ABB RobotStudio station: Final_Project.rspag

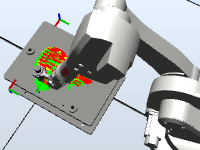
--- station ---
Station Final_Project (saved by RobotStudio 6.6.7603.115)
Controller IRB_1600_8kg_1.45m
  mechanical unit ROB_1: IRB1600_8_145__02, 6 joints, base frame (0, 0, 0) mm
Layout (positions relative to the parent item):
  - IRB1600_8_145__02 [mechanism, from Robots\IRB1600_8_145_G_02.rslib] at (0, 0, 0) mm; joint values [0.2552, 0.6803, 0.4832, 0.5846, -0.2854, -0.363] (rad or m)
  - Robotpedestal1400_H240 [part, from Equipment\Robot Pedestal 1400 H240.rslib] at (876.55, 58.92, 0) mm
  - MyTool [mechanism, from Training Objects\myTool.rslib] at (841.22, 209, 428.53) mm, rotated rx 180 ry 38 rz 180 deg
Attachment: MyTool is attached to IRB1600_8_145__02 / Link6

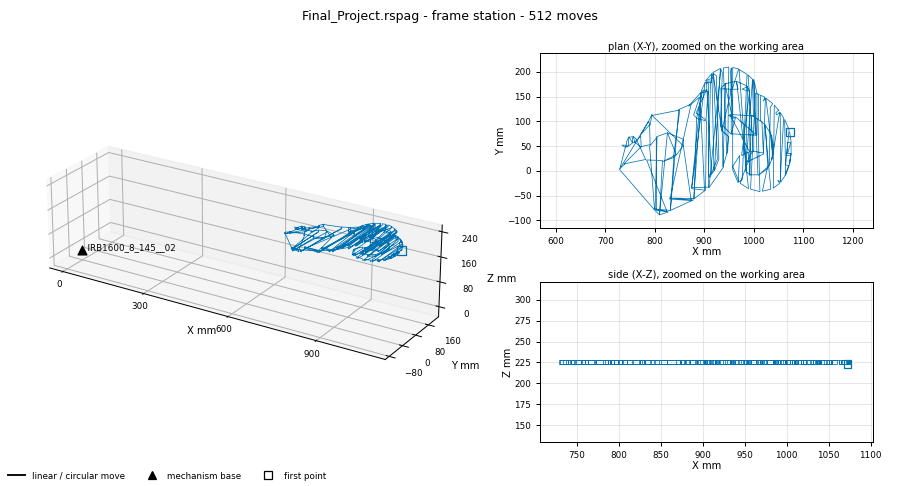
[picture p0: tool path of Final_Project.rspag in frame station, 512 of 512 moves have a stored position in this frame; points joined in program order, loops and branches not executed]
--- Backups/IRB_1600_8kg_1.45m/RAPID/TASK1/PROGMOD/CalibData.mod ---
MODULE CalibData
	TASK PERS wobjdata Workobject_1:=[FALSE,TRUE,"",[[1116.549,-245,225],[0.707106781,0,0,0.707106781]],[[600,0,8],[0,0,1,0]]];
	TASK PERS tooldata MyTool:=[TRUE,[[31.792631019,0,229.638935148],[0.945518576,0,0.325568154,0]],[1,[0,0,1],[1,0,0,0],0,0,0]];
ENDMODULE

--- Backups/IRB_1600_8kg_1.45m/RAPID/TASK1/PROGMOD/Module1.mod ---
MODULE Module1
    CONST robtarget point_0_clearance:=[[277,44,10],[0.707106781,0,0,0.707106781],[0,0,-1,1],[9E+09,9E+09,9E+09,9E+09,9E+09,9E+09]];
    CONST robtarget point_0_contact:=[[277,44,5],[0.707106781,0,0,0.707106781],[0,0,-1,1],[9E+09,9E+09,9E+09,9E+09,9E+09,9E+09]];
    CONST robtarget point_1_contact:=[[296,41,5],[0.707106781,0,0,0.707106781],[0,0,-1,1],[9E+09,9E+09,9E+09,9E+09,9E+09,9E+09]];
    CONST robtarget point_1_clearance:=[[296,41,10],[0.707106781,0,0,0.707106781],[0,0,-1,1],[9E+09,9E+09,9E+09,9E+09,9E+09,9E+09]];
    CONST robtarget point_2_clearance:=[[322,41,10],[0.707106781,0,0,0.707106781],[0,0,-1,1],[9E+09,9E+09,9E+09,9E+09,9E+09,9E+09]];
    CONST robtarget point_2_contact:=[[322,41,5],[0.707106781,0,0,0.707106781],[0,0,-1,1],[9E+09,9E+09,9E+09,9E+09,9E+09,9E+09]];
    CONST robtarget point_3_contact:=[[341,44,5],[0.707106781,0,0,0.707106781],[0,0,-1,1],[9E+09,9E+09,9E+09,9E+09,9E+09,9E+09]];
    CONST robtarget point_3_clearance:=[[341,44,10],[0.707106781,0,0,0.707106781],[0,0,-1,1],[9E+09,9E+09,9E+09,9E+09,9E+09,9E+09]];
    CONST robtarget point_4_clearance:=[[320,41,10],[0.707106781,0,0,0.707106781],[0,0,-1,1],[9E+09,9E+09,9E+09,9E+09,9E+09,9E+09]];
    CONST robtarget point_4_contact:=[[320,41,5],[0.707106781,0,0,0.707106781],[0,0,-1,1],[9E+09,9E+09,9E+09,9E+09,9E+09,9E+09]];
    CONST robtarget point_5_contact:=[[320,48,5],[0.707106781,0,0,0.707106781],[0,0,-1,1],[9E+09,9E+09,9E+09,9E+09,9E+09,9E+09]];
    CONST robtarget point_5_clearance:=[[320,48,10],[0.707106781,0,0,0.707106781],[0,0,-1,1],[9E+09,9E+09,9E+09,9E+09,9E+09,9E+09]];
    CONST robtarget point_6_clearance:=[[298,42,10],[0.707106781,0,0,0.707106781],[0,0,-1,1],[9E+09,9E+09,9E+09,9E+09,9E+09,9E+09]];
    CONST robtarget point_6_contact:=[[298,42,5],[0.707106781,0,0,0.707106781],[0,0,-1,1],[9E+09,9E+09,9E+09,9E+09,9E+09,9E+09]];
    CONST robtarget point_7_contact:=[[298,48,5],[0.707106781,0,0,0.707106781],[0,0,-1,1],[9E+09,9E+09,9E+09,9E+09,9E+09,9E+09]];
    CONST robtarget point_7_clearance:=[[298,48,10],[0.707106781,0,0,0.707106781],[0,0,-1,1],[9E+09,9E+09,9E+09,9E+09,9E+09,9E+09]];
    CONST robtarget point_8_clearance:=[[324,50,10],[0.707106781,0,0,0.707106781],[0,0,-1,1],[9E+09,9E+09,9E+09,9E+09,9E+09,9E+09]];
    CONST robtarget point_8_contact:=[[324,50,5],[0.707106781,0,0,0.707106781],[0,0,-1,1],[9E+09,9E+09,9E+09,9E+09,9E+09,9E+09]];
    CONST robtarget point_9_contact:=[[323,42,5],[0.707106781,0,0,0.707106781],[0,0,-1,1],[9E+09,9E+09,9E+09,9E+09,9E+09,9E+09]];
    CONST robtarget point_9_clearance:=[[323,42,10],[0.707106781,0,0,0.707106781],[0,0,-1,1],[9E+09,9E+09,9E+09,9E+09,9E+09,9E+09]];
    CONST robtarget point_10_clearance:=[[345,45,10],[0.707106781,0,0,0.707106781],[0,0,-1,1],[9E+09,9E+09,9E+09,9E+09,9E+09,9E+09]];
    CONST robtarget point_10_contact:=[[345,45,5],[0.707106781,0,0,0.707106781],[0,0,-1,1],[9E+09,9E+09,9E+09,9E+09,9E+09,9E+09]];
    CONST robtarget point_11_contact:=[[364,52,5],[0.707106781,0,0,0.707106781],[-1,-1,0,1],[9E+09,9E+09,9E+09,9E+09,9E+09,9E+09]];
    CONST robtarget point_11_clearance:=[[364,52,10],[0.707106781,0,0,0.707106781],[-1,-1,0,1],[9E+09,9E+09,9E+09,9E+09,9E+09,9E+09]];
    CONST robtarget point_12_clearance:=[[251,54,10],[0.707106781,0,0,0.707106781],[0,0,-1,1],[9E+09,9E+09,9E+09,9E+09,9E+09,9E+09]];
    CONST robtarget point_12_contact:=[[251,54,5],[0.707106781,0,0,0.707106781],[0,0,-1,1],[9E+09,9E+09,9E+09,9E+09,9E+09,9E+09]];
    CONST robtarget point_13_contact:=[[272,45,5],[0.707106781,0,0,0.707106781],[0,0,-1,1],[9E+09,9E+09,9E+09,9E+09,9E+09,9E+09]];
    CONST robtarget point_13_clearance:=[[272,45,10],[0.707106781,0,0,0.707106781],[0,0,-1,1],[9E+09,9E+09,9E+09,9E+09,9E+09,9E+09]];
    CONST robtarget point_14_clearance:=[[343,52,10],[0.707106781,0,0,0.707106781],[0,0,-1,1],[9E+09,9E+09,9E+09,9E+09,9E+09,9E+09]];
    CONST robtarget point_14_contact:=[[343,52,5],[0.707106781,0,0,0.707106781],[0,0,-1,1],[9E+09,9E+09,9E+09,9E+09,9E+09,9E+09]];
    CONST robtarget point_15_contact:=[[344,46,5],[0.707106781,0,0,0.707106781],[0,0,-1,1],[9E+09,9E+09,9E+09,9E+09,9E+09,9E+09]];
    CONST robtarget point_15_clearance:=[[344,46,10],[0.707106781,0,0,0.707106781],[0,0,-1,1],[9E+09,9E+09,9E+09,9E+09,9E+09,9E+09]];
    CONST robtarget point_16_clearance:=[[366,54,10],[0.707106781,0,0,0.707106781],[-1,-1,0,1],[9E+09,9E+09,9E+09,9E+09,9E+09,9E+09]];
    CONST robtarget point_16_contact:=[[366,54,5],[0.707106781,0,0,0.707106781],[-1,-1,0,1],[9E+09,9E+09,9E+09,9E+09,9E+09,9E+09]];
    CONST robtarget point_17_contact:=[[378,62,5],[0.707106781,0,0,0.707106781],[-1,-1,0,1],[9E+09,9E+09,9E+09,9E+09,9E+09,9E+09]];
    CONST robtarget point_17_clearance:=[[378,62,10],[0.707106781,0,0,0.707106781],[-1,-1,0,1],[9E+09,9E+09,9E+09,9E+09,9E+09,9E+09]];
    CONST robtarget point_18_clearance:=[[237,63,10],[0.707106781,0,0,0.707106781],[0,0,-1,1],[9E+09,9E+09,9E+09,9E+09,9E+09,9E+09]];
    CONST robtarget point_18_contact:=[[237,63,5],[0.707106781,0,0,0.707106781],[0,0,-1,1],[9E+09,9E+09,9E+09,9E+09,9E+09,9E+09]];
    CONST robtarget point_19_contact:=[[248,56,5],[0.707106781,0,0,0.707106781],[0,0,-1,1],[9E+09,9E+09,9E+09,9E+09,9E+09,9E+09]];
    CONST robtarget point_19_clearance:=[[248,56,10],[0.707106781,0,0,0.707106781],[0,0,-1,1],[9E+09,9E+09,9E+09,9E+09,9E+09,9E+09]];
    CONST robtarget point_20_clearance:=[[377,63,10],[0.707106781,0,0,0.707106781],[-1,-1,0,1],[9E+09,9E+09,9E+09,9E+09,9E+09,9E+09]];
    CONST robtarget point_20_contact:=[[377,63,5],[0.707106781,0,0,0.707106781],[-1,-1,0,1],[9E+09,9E+09,9E+09,9E+09,9E+09,9E+09]];
    CONST robtarget point_21_contact:=[[374,68,5],[0.707106781,0,0,0.707106781],[-1,-1,0,1],[9E+09,9E+09,9E+09,9E+09,9E+09,9E+09]];
    CONST robtarget point_21_clearance:=[[374,68,10],[0.707106781,0,0,0.707106781],[-1,-1,0,1],[9E+09,9E+09,9E+09,9E+09,9E+09,9E+09]];
    CONST robtarget point_22_clearance:=[[380,64,10],[0.707106781,0,0,0.707106781],[-1,-1,0,1],[9E+09,9E+09,9E+09,9E+09,9E+09,9E+09]];
    CONST robtarget point_22_contact:=[[380,64,5],[0.707106781,0,0,0.707106781],[-1,-1,0,1],[9E+09,9E+09,9E+09,9E+09,9E+09,9E+09]];
    CONST robtarget point_23_contact:=[[390,77,5],[0.707106781,0,0,0.707106781],[-1,-1,0,1],[9E+09,9E+09,9E+09,9E+09,9E+09,9E+09]];
    CONST robtarget point_23_clearance:=[[390,77,10],[0.707106781,0,0,0.707106781],[-1,-1,0,1],[9E+09,9E+09,9E+09,9E+09,9E+09,9E+09]];
    CONST robtarget point_24_clearance:=[[222,75,10],[0.707106781,0,0,0.707106781],[0,0,-1,1],[9E+09,9E+09,9E+09,9E+09,9E+09,9E+09]];
    CONST robtarget point_24_contact:=[[222,75,5],[0.707106781,0,0,0.707106781],[0,0,-1,1],[9E+09,9E+09,9E+09,9E+09,9E+09,9E+09]];
    CONST robtarget point_25_contact:=[[233,66,5],[0.707106781,0,0,0.707106781],[0,0,-1,1],[9E+09,9E+09,9E+09,9E+09,9E+09,9E+09]];
    CONST robtarget point_25_clearance:=[[233,66,10],[0.707106781,0,0,0.707106781],[0,0,-1,1],[9E+09,9E+09,9E+09,9E+09,9E+09,9E+09]];
    CONST robtarget point_26_clearance:=[[232,66,10],[0.707106781,0,0,0.707106781],[0,0,-1,1],[9E+09,9E+09,9E+09,9E+09,9E+09,9E+09]];
    CONST robtarget point_26_contact:=[[232,66,5],[0.707106781,0,0,0.707106781],[0,0,-1,1],[9E+09,9E+09,9E+09,9E+09,9E+09,9E+09]];
    CONST robtarget point_27_contact:=[[238,72,5],[0.707106781,0,0,0.707106781],[0,0,-1,1],[9E+09,9E+09,9E+09,9E+09,9E+09,9E+09]];
    CONST robtarget point_27_clearance:=[[238,72,10],[0.707106781,0,0,0.707106781],[0,0,-1,1],[9E+09,9E+09,9E+09,9E+09,9E+09,9E+09]];
    CONST robtarget point_28_clearance:=[[242,70,10],[0.707106781,0,0,0.707106781],[0,0,-1,1],[9E+09,9E+09,9E+09,9E+09,9E+09,9E+09]];
    CONST robtarget point_28_contact:=[[242,70,5],[0.707106781,0,0,0.707106781],[0,0,-1,1],[9E+09,9E+09,9E+09,9E+09,9E+09,9E+09]];
    CONST robtarget point_29_contact:=[[236,64,5],[0.707106781,0,0,0.707106781],[0,0,-1,1],[9E+09,9E+09,9E+09,9E+09,9E+09,9E+09]];
    CONST robtarget point_29_clearance:=[[236,64,10],[0.707106781,0,0,0.707106781],[0,0,-1,1],[9E+09,9E+09,9E+09,9E+09,9E+09,9E+09]];
    CONST robtarget point_30_clearance:=[[310,76,10],[0.707106781,0,0,0.707106781],[0,0,-1,1],[9E+09,9E+09,9E+09,9E+09,9E+09,9E+09]];
    CONST robtarget point_30_contact:=[[310,76,5],[0.707106781,0,0,0.707106781],[0,0,-1,1],[9E+09,9E+09,9E+09,9E+09,9E+09,9E+09]];
    CONST robtarget point_31_contact:=[[283,81,5],[0.707106781,0,0,0.707106781],[0,0,-1,1],[9E+09,9E+09,9E+09,9E+09,9E+09,9E+09]];
    CONST robtarget point_31_clearance:=[[283,81,10],[0.707106781,0,0,0.707106781],[0,0,-1,1],[9E+09,9E+09,9E+09,9E+09,9E+09,9E+09]];
    CONST robtarget point_32_clearance:=[[323,78,10],[0.707106781,0,0,0.707106781],[0,0,-1,1],[9E+09,9E+09,9E+09,9E+09,9E+09,9E+09]];
    CONST robtarget point_32_contact:=[[323,78,5],[0.707106781,0,0,0.707106781],[0,0,-1,1],[9E+09,9E+09,9E+09,9E+09,9E+09,9E+09]];
    CONST robtarget point_33_contact:=[[310,77,5],[0.707106781,0,0,0.707106781],[0,0,-1,1],[9E+09,9E+09,9E+09,9E+09,9E+09,9E+09]];
    CONST robtarget point_33_clearance:=[[310,77,10],[0.707106781,0,0,0.707106781],[0,0,-1,1],[9E+09,9E+09,9E+09,9E+09,9E+09,9E+09]];
    CONST robtarget point_34_clearance:=[[332,80,10],[0.707106781,0,0,0.707106781],[0,0,-1,1],[9E+09,9E+09,9E+09,9E+09,9E+09,9E+09]];
    CONST robtarget point_34_contact:=[[332,80,5],[0.707106781,0,0,0.707106781],[0,0,-1,1],[9E+09,9E+09,9E+09,9E+09,9E+09,9E+09]];
    CONST robtarget point_35_contact:=[[321,78,5],[0.707106781,0,0,0.707106781],[0,0,-1,1],[9E+09,9E+09,9E+09,9E+09,9E+09,9E+09]];
    CONST robtarget point_35_clearance:=[[321,78,10],[0.707106781,0,0,0.707106781],[0,0,-1,1],[9E+09,9E+09,9E+09,9E+09,9E+09,9E+09]];
    CONST robtarget point_36_clearance:=[[208,92,10],[0.707106781,0,0,0.707106781],[0,0,-1,1],[9E+09,9E+09,9E+09,9E+09,9E+09,9E+09]];
    CONST robtarget point_36_contact:=[[208,92,5],[0.707106781,0,0,0.707106781],[0,0,-1,1],[9E+09,9E+09,9E+09,9E+09,9E+09,9E+09]];
    CONST robtarget point_37_contact:=[[219,78,5],[0.707106781,0,0,0.707106781],[0,0,-1,1],[9E+09,9E+09,9E+09,9E+09,9E+09,9E+09]];
    CONST robtarget point_37_clearance:=[[219,78,10],[0.707106781,0,0,0.707106781],[0,0,-1,1],[9E+09,9E+09,9E+09,9E+09,9E+09,9E+09]];
    CONST robtarget point_38_clearance:=[[219,78,10],[0.707106781,0,0,0.707106781],[0,0,-1,1],[9E+09,9E+09,9E+09,9E+09,9E+09,9E+09]];
    CONST robtarget point_38_contact:=[[219,78,5],[0.707106781,0,0,0.707106781],[0,0,-1,1],[9E+09,9E+09,9E+09,9E+09,9E+09,9E+09]];
    CONST robtarget point_39_contact:=[[226,83,5],[0.707106781,0,0,0.707106781],[0,0,-1,1],[9E+09,9E+09,9E+09,9E+09,9E+09,9E+09]];
    CONST robtarget point_39_clearance:=[[226,83,10],[0.707106781,0,0,0.707106781],[0,0,-1,1],[9E+09,9E+09,9E+09,9E+09,9E+09,9E+09]];
    CONST robtarget point_40_clearance:=[[344,85,10],[0.707106781,0,0,0.707106781],[0,0,-1,1],[9E+09,9E+09,9E+09,9E+09,9E+09,9E+09]];
    CONST robtarget point_40_contact:=[[344,85,5],[0.707106781,0,0,0.707106781],[0,0,-1,1],[9E+09,9E+09,9E+09,9E+09,9E+09,9E+09]];
    CONST robtarget point_41_contact:=[[329,79,5],[0.707106781,0,0,0.707106781],[0,0,-1,1],[9E+09,9E+09,9E+09,9E+09,9E+09,9E+09]];
    CONST robtarget point_41_clearance:=[[329,79,10],[0.707106781,0,0,0.707106781],[0,0,-1,1],[9E+09,9E+09,9E+09,9E+09,9E+09,9E+09]];
    CONST robtarget point_42_clearance:=[[284,80,10],[0.707106781,0,0,0.707106781],[0,0,-1,1],[9E+09,9E+09,9E+09,9E+09,9E+09,9E+09]];
    CONST robtarget point_42_contact:=[[284,80,5],[0.707106781,0,0,0.707106781],[0,0,-1,1],[9E+09,9E+09,9E+09,9E+09,9E+09,9E+09]];
    CONST robtarget point_43_contact:=[[261,94,5],[0.707106781,0,0,0.707106781],[0,0,-1,1],[9E+09,9E+09,9E+09,9E+09,9E+09,9E+09]];
    CONST robtarget point_43_clearance:=[[261,94,10],[0.707106781,0,0,0.707106781],[0,0,-1,1],[9E+09,9E+09,9E+09,9E+09,9E+09,9E+09]];
    CONST robtarget point_44_clearance:=[[392,82,10],[0.707106781,0,0,0.707106781],[-1,-1,0,1],[9E+09,9E+09,9E+09,9E+09,9E+09,9E+09]];
    CONST robtarget point_44_contact:=[[392,82,5],[0.707106781,0,0,0.707106781],[-1,-1,0,1],[9E+09,9E+09,9E+09,9E+09,9E+09,9E+09]];
    CONST robtarget point_45_contact:=[[396,99,5],[0.707106781,0,0,0.707106781],[-1,-1,0,1],[9E+09,9E+09,9E+09,9E+09,9E+09,9E+09]];
    CONST robtarget point_45_clearance:=[[396,99,10],[0.707106781,0,0,0.707106781],[-1,-1,0,1],[9E+09,9E+09,9E+09,9E+09,9E+09,9E+09]];
    CONST robtarget point_46_clearance:=[[349,89,10],[0.707106781,0,0,0.707106781],[0,0,-1,1],[9E+09,9E+09,9E+09,9E+09,9E+09,9E+09]];
    CONST robtarget point_46_contact:=[[349,89,5],[0.707106781,0,0,0.707106781],[0,0,-1,1],[9E+09,9E+09,9E+09,9E+09,9E+09,9E+09]];
    CONST robtarget point_47_contact:=[[344,85,5],[0.707106781,0,0,0.707106781],[0,0,-1,1],[9E+09,9E+09,9E+09,9E+09,9E+09,9E+09]];
    CONST robtarget point_47_clearance:=[[344,85,10],[0.707106781,0,0,0.707106781],[0,0,-1,1],[9E+09,9E+09,9E+09,9E+09,9E+09,9E+09]];
    CONST robtarget point_48_clearance:=[[364,107,10],[0.707106781,0,0,0.707106781],[-1,-1,0,1],[9E+09,9E+09,9E+09,9E+09,9E+09,9E+09]];
    CONST robtarget point_48_contact:=[[364,107,5],[0.707106781,0,0,0.707106781],[-1,-1,0,1],[9E+09,9E+09,9E+09,9E+09,9E+09,9E+09]];
    CONST robtarget point_49_contact:=[[350,88,5],[0.707106781,0,0,0.707106781],[0,0,-1,1],[9E+09,9E+09,9E+09,9E+09,9E+09,9E+09]];
    CONST robtarget point_49_clearance:=[[350,88,10],[0.707106781,0,0,0.707106781],[0,0,-1,1],[9E+09,9E+09,9E+09,9E+09,9E+09,9E+09]];
    CONST robtarget point_50_clearance:=[[263,93,10],[0.707106781,0,0,0.707106781],[0,0,-1,1],[9E+09,9E+09,9E+09,9E+09,9E+09,9E+09]];
    CONST robtarget point_50_contact:=[[263,93,5],[0.707106781,0,0,0.707106781],[0,0,-1,1],[9E+09,9E+09,9E+09,9E+09,9E+09,9E+09]];
    CONST robtarget point_51_contact:=[[253,103,5],[0.707106781,0,0,0.707106781],[0,0,-1,1],[9E+09,9E+09,9E+09,9E+09,9E+09,9E+09]];
    CONST robtarget point_51_clearance:=[[253,103,10],[0.707106781,0,0,0.707106781],[0,0,-1,1],[9E+09,9E+09,9E+09,9E+09,9E+09,9E+09]];
    CONST robtarget point_52_clearance:=[[202,103,10],[0.707106781,0,0,0.707106781],[0,0,-1,1],[9E+09,9E+09,9E+09,9E+09,9E+09,9E+09]];
    CONST robtarget point_52_contact:=[[202,103,5],[0.707106781,0,0,0.707106781],[0,0,-1,1],[9E+09,9E+09,9E+09,9E+09,9E+09,9E+09]];
    CONST robtarget point_53_contact:=[[206,94,5],[0.707106781,0,0,0.707106781],[0,0,-1,1],[9E+09,9E+09,9E+09,9E+09,9E+09,9E+09]];
    CONST robtarget point_53_clearance:=[[206,94,10],[0.707106781,0,0,0.707106781],[0,0,-1,1],[9E+09,9E+09,9E+09,9E+09,9E+09,9E+09]];
    CONST robtarget point_54_clearance:=[[214,97,10],[0.707106781,0,0,0.707106781],[0,0,-1,1],[9E+09,9E+09,9E+09,9E+09,9E+09,9E+09]];
    CONST robtarget point_54_contact:=[[214,97,5],[0.707106781,0,0,0.707106781],[0,0,-1,1],[9E+09,9E+09,9E+09,9E+09,9E+09,9E+09]];
    CONST robtarget point_55_contact:=[[208,93,5],[0.707106781,0,0,0.707106781],[0,0,-1,1],[9E+09,9E+09,9E+09,9E+09,9E+09,9E+09]];
    CONST robtarget point_55_clearance:=[[208,93,10],[0.707106781,0,0,0.707106781],[0,0,-1,1],[9E+09,9E+09,9E+09,9E+09,9E+09,9E+09]];
    CONST robtarget point_56_clearance:=[[321,97,10],[0.707106781,0,0,0.707106781],[0,0,-1,1],[9E+09,9E+09,9E+09,9E+09,9E+09,9E+09]];
    CONST robtarget point_56_contact:=[[321,97,5],[0.707106781,0,0,0.707106781],[0,0,-1,1],[9E+09,9E+09,9E+09,9E+09,9E+09,9E+09]];
    CONST robtarget point_57_contact:=[[337,130,5],[0.707106781,0,0,0.707106781],[0,0,-1,1],[9E+09,9E+09,9E+09,9E+09,9E+09,9E+09]];
    CONST robtarget point_57_clearance:=[[337,130,10],[0.707106781,0,0,0.707106781],[0,0,-1,1],[9E+09,9E+09,9E+09,9E+09,9E+09,9E+09]];
    CONST robtarget point_58_clearance:=[[315,119,10],[0.707106781,0,0,0.707106781],[0,0,-1,1],[9E+09,9E+09,9E+09,9E+09,9E+09,9E+09]];
    CONST robtarget point_58_contact:=[[315,119,5],[0.707106781,0,0,0.707106781],[0,0,-1,1],[9E+09,9E+09,9E+09,9E+09,9E+09,9E+09]];
    CONST robtarget point_59_contact:=[[319,97,5],[0.707106781,0,0,0.707106781],[0,0,-1,1],[9E+09,9E+09,9E+09,9E+09,9E+09,9E+09]];
    CONST robtarget point_59_clearance:=[[319,97,10],[0.707106781,0,0,0.707106781],[0,0,-1,1],[9E+09,9E+09,9E+09,9E+09,9E+09,9E+09]];
    CONST robtarget point_60_clearance:=[[256,100,10],[0.707106781,0,0,0.707106781],[0,0,-1,1],[9E+09,9E+09,9E+09,9E+09,9E+09,9E+09]];
    CONST robtarget point_60_contact:=[[256,100,5],[0.707106781,0,0,0.707106781],[0,0,-1,1],[9E+09,9E+09,9E+09,9E+09,9E+09,9E+09]];
    CONST robtarget point_61_contact:=[[251,108,5],[0.707106781,0,0,0.707106781],[0,0,-1,1],[9E+09,9E+09,9E+09,9E+09,9E+09,9E+09]];
    CONST robtarget point_61_clearance:=[[251,108,10],[0.707106781,0,0,0.707106781],[0,0,-1,1],[9E+09,9E+09,9E+09,9E+09,9E+09,9E+09]];
    CONST robtarget point_62_clearance:=[[397,104,10],[0.707106781,0,0,0.707106781],[-1,-1,0,1],[9E+09,9E+09,9E+09,9E+09,9E+09,9E+09]];
    CONST robtarget point_62_contact:=[[397,104,5],[0.707106781,0,0,0.707106781],[-1,-1,0,1],[9E+09,9E+09,9E+09,9E+09,9E+09,9E+09]];
    CONST robtarget point_63_contact:=[[392,123,5],[0.707106781,0,0,0.707106781],[-1,-1,0,1],[9E+09,9E+09,9E+09,9E+09,9E+09,9E+09]];
    CONST robtarget point_63_clearance:=[[392,123,10],[0.707106781,0,0,0.707106781],[-1,-1,0,1],[9E+09,9E+09,9E+09,9E+09,9E+09,9E+09]];
    CONST robtarget point_64_clearance:=[[198,113,10],[0.707106781,0,0,0.707106781],[0,0,-1,1],[9E+09,9E+09,9E+09,9E+09,9E+09,9E+09]];
    CONST robtarget point_64_contact:=[[198,113,5],[0.707106781,0,0,0.707106781],[0,0,-1,1],[9E+09,9E+09,9E+09,9E+09,9E+09,9E+09]];
    CONST robtarget point_65_contact:=[[201,105,5],[0.707106781,0,0,0.707106781],[0,0,-1,1],[9E+09,9E+09,9E+09,9E+09,9E+09,9E+09]];
    CONST robtarget point_65_clearance:=[[201,105,10],[0.707106781,0,0,0.707106781],[0,0,-1,1],[9E+09,9E+09,9E+09,9E+09,9E+09,9E+09]];
    CONST robtarget point_66_clearance:=[[202,107,10],[0.707106781,0,0,0.707106781],[0,0,-1,1],[9E+09,9E+09,9E+09,9E+09,9E+09,9E+09]];
    CONST robtarget point_66_contact:=[[202,107,5],[0.707106781,0,0,0.707106781],[0,0,-1,1],[9E+09,9E+09,9E+09,9E+09,9E+09,9E+09]];
    CONST robtarget point_67_contact:=[[208,107,5],[0.707106781,0,0,0.707106781],[0,0,-1,1],[9E+09,9E+09,9E+09,9E+09,9E+09,9E+09]];
    CONST robtarget point_67_clearance:=[[208,107,10],[0.707106781,0,0,0.707106781],[0,0,-1,1],[9E+09,9E+09,9E+09,9E+09,9E+09,9E+09]];
    CONST robtarget point_68_clearance:=[[251,107,10],[0.707106781,0,0,0.707106781],[0,0,-1,1],[9E+09,9E+09,9E+09,9E+09,9E+09,9E+09]];
    CONST robtarget point_68_contact:=[[251,107,5],[0.707106781,0,0,0.707106781],[0,0,-1,1],[9E+09,9E+09,9E+09,9E+09,9E+09,9E+09]];
    CONST robtarget point_69_contact:=[[243,121,5],[0.707106781,0,0,0.707106781],[0,0,-1,1],[9E+09,9E+09,9E+09,9E+09,9E+09,9E+09]];
    CONST robtarget point_69_clearance:=[[243,121,10],[0.707106781,0,0,0.707106781],[0,0,-1,1],[9E+09,9E+09,9E+09,9E+09,9E+09,9E+09]];
    CONST robtarget point_70_clearance:=[[363,125,10],[0.707106781,0,0,0.707106781],[-1,-1,0,1],[9E+09,9E+09,9E+09,9E+09,9E+09,9E+09]];
    CONST robtarget point_70_contact:=[[363,125,5],[0.707106781,0,0,0.707106781],[-1,-1,0,1],[9E+09,9E+09,9E+09,9E+09,9E+09,9E+09]];
    CONST robtarget point_71_contact:=[[363,108,5],[0.707106781,0,0,0.707106781],[-1,-1,0,1],[9E+09,9E+09,9E+09,9E+09,9E+09,9E+09]];
    CONST robtarget point_71_clearance:=[[363,108,10],[0.707106781,0,0,0.707106781],[-1,-1,0,1],[9E+09,9E+09,9E+09,9E+09,9E+09,9E+09]];
    CONST robtarget point_72_clearance:=[[172,116,10],[0.707106781,0,0,0.707106781],[0,0,-1,1],[9E+09,9E+09,9E+09,9E+09,9E+09,9E+09]];
    CONST robtarget point_72_contact:=[[172,116,5],[0.707106781,0,0,0.707106781],[0,0,-1,1],[9E+09,9E+09,9E+09,9E+09,9E+09,9E+09]];
    CONST robtarget point_73_contact:=[[198,110,5],[0.707106781,0,0,0.707106781],[0,0,-1,1],[9E+09,9E+09,9E+09,9E+09,9E+09,9E+09]];
    CONST robtarget point_73_clearance:=[[198,110,10],[0.707106781,0,0,0.707106781],[0,0,-1,1],[9E+09,9E+09,9E+09,9E+09,9E+09,9E+09]];
    CONST robtarget point_74_clearance:=[[283,110,10],[0.707106781,0,0,0.707106781],[0,0,-1,1],[9E+09,9E+09,9E+09,9E+09,9E+09,9E+09]];
    CONST robtarget point_74_contact:=[[283,110,5],[0.707106781,0,0,0.707106781],[0,0,-1,1],[9E+09,9E+09,9E+09,9E+09,9E+09,9E+09]];
    CONST robtarget point_75_contact:=[[280,162,5],[0.707106781,0,0,0.707106781],[0,0,-1,1],[9E+09,9E+09,9E+09,9E+09,9E+09,9E+09]];
    CONST robtarget point_75_clearance:=[[280,162,10],[0.707106781,0,0,0.707106781],[0,0,-1,1],[9E+09,9E+09,9E+09,9E+09,9E+09,9E+09]];
    CONST robtarget point_76_clearance:=[[246,153,10],[0.707106781,0,0,0.707106781],[0,0,-1,1],[9E+09,9E+09,9E+09,9E+09,9E+09,9E+09]];
    CONST robtarget point_76_contact:=[[246,153,5],[0.707106781,0,0,0.707106781],[0,0,-1,1],[9E+09,9E+09,9E+09,9E+09,9E+09,9E+09]];
    CONST robtarget point_77_contact:=[[281,113,5],[0.707106781,0,0,0.707106781],[0,0,-1,1],[9E+09,9E+09,9E+09,9E+09,9E+09,9E+09]];
    CONST robtarget point_77_clearance:=[[281,113,10],[0.707106781,0,0,0.707106781],[0,0,-1,1],[9E+09,9E+09,9E+09,9E+09,9E+09,9E+09]];
    CONST robtarget point_78_clearance:=[[170,117,10],[0.707106781,0,0,0.707106781],[0,0,-1,1],[9E+09,9E+09,9E+09,9E+09,9E+09,9E+09]];
    CONST robtarget point_78_contact:=[[170,117,5],[0.707106781,0,0,0.707106781],[0,0,-1,1],[9E+09,9E+09,9E+09,9E+09,9E+09,9E+09]];
    CONST robtarget point_79_contact:=[[173,119,5],[0.707106781,0,0,0.707106781],[0,0,-1,1],[9E+09,9E+09,9E+09,9E+09,9E+09,9E+09]];
    CONST robtarget point_79_clearance:=[[173,119,10],[0.707106781,0,0,0.707106781],[0,0,-1,1],[9E+09,9E+09,9E+09,9E+09,9E+09,9E+09]];
    CONST robtarget point_80_clearance:=[[244,117,10],[0.707106781,0,0,0.707106781],[0,0,-1,1],[9E+09,9E+09,9E+09,9E+09,9E+09,9E+09]];
    CONST robtarget point_80_contact:=[[244,117,5],[0.707106781,0,0,0.707106781],[0,0,-1,1],[9E+09,9E+09,9E+09,9E+09,9E+09,9E+09]];
    CONST robtarget point_81_contact:=[[241,165,5],[0.707106781,0,0,0.707106781],[0,0,-1,1],[9E+09,9E+09,9E+09,9E+09,9E+09,9E+09]];
    CONST robtarget point_81_clearance:=[[241,165,10],[0.707106781,0,0,0.707106781],[0,0,-1,1],[9E+09,9E+09,9E+09,9E+09,9E+09,9E+09]];
    CONST robtarget point_82_clearance:=[[316,125,10],[0.707106781,0,0,0.707106781],[0,0,-1,1],[9E+09,9E+09,9E+09,9E+09,9E+09,9E+09]];
    CONST robtarget point_82_contact:=[[316,125,5],[0.707106781,0,0,0.707106781],[0,0,-1,1],[9E+09,9E+09,9E+09,9E+09,9E+09,9E+09]];
    CONST robtarget point_83_contact:=[[316,117,5],[0.707106781,0,0,0.707106781],[0,0,-1,1],[9E+09,9E+09,9E+09,9E+09,9E+09,9E+09]];
    CONST robtarget point_83_clearance:=[[316,117,10],[0.707106781,0,0,0.707106781],[0,0,-1,1],[9E+09,9E+09,9E+09,9E+09,9E+09,9E+09]];
    CONST robtarget point_84_clearance:=[[161,128,10],[0.707106781,0,0,0.707106781],[0,0,-1,1],[9E+09,9E+09,9E+09,9E+09,9E+09,9E+09]];
    CONST robtarget point_84_contact:=[[161,128,5],[0.707106781,0,0,0.707106781],[0,0,-1,1],[9E+09,9E+09,9E+09,9E+09,9E+09,9E+09]];
    CONST robtarget point_85_contact:=[[170,119,5],[0.707106781,0,0,0.707106781],[0,0,-1,1],[9E+09,9E+09,9E+09,9E+09,9E+09,9E+09]];
    CONST robtarget point_85_clearance:=[[170,119,10],[0.707106781,0,0,0.707106781],[0,0,-1,1],[9E+09,9E+09,9E+09,9E+09,9E+09,9E+09]];
    CONST robtarget point_86_clearance:=[[355,133,10],[0.707106781,0,0,0.707106781],[0,-1,0,1],[9E+09,9E+09,9E+09,9E+09,9E+09,9E+09]];
    CONST robtarget point_86_contact:=[[355,133,5],[0.707106781,0,0,0.707106781],[0,-1,0,1],[9E+09,9E+09,9E+09,9E+09,9E+09,9E+09]];
    CONST robtarget point_87_contact:=[[364,124,5],[0.707106781,0,0,0.707106781],[-1,-1,0,1],[9E+09,9E+09,9E+09,9E+09,9E+09,9E+09]];
    CONST robtarget point_87_clearance:=[[364,124,10],[0.707106781,0,0,0.707106781],[-1,-1,0,1],[9E+09,9E+09,9E+09,9E+09,9E+09,9E+09]];
    CONST robtarget point_88_clearance:=[[193,125,10],[0.707106781,0,0,0.707106781],[0,0,-1,1],[9E+09,9E+09,9E+09,9E+09,9E+09,9E+09]];
    CONST robtarget point_88_contact:=[[193,125,5],[0.707106781,0,0,0.707106781],[0,0,-1,1],[9E+09,9E+09,9E+09,9E+09,9E+09,9E+09]];
    CONST robtarget point_89_contact:=[[185,130,5],[0.707106781,0,0,0.707106781],[0,0,-1,1],[9E+09,9E+09,9E+09,9E+09,9E+09,9E+09]];
    CONST robtarget point_89_clearance:=[[185,130,10],[0.707106781,0,0,0.707106781],[0,0,-1,1],[9E+09,9E+09,9E+09,9E+09,9E+09,9E+09]];
    CONST robtarget point_90_clearance:=[[190,140,10],[0.707106781,0,0,0.707106781],[0,0,-1,1],[9E+09,9E+09,9E+09,9E+09,9E+09,9E+09]];
    CONST robtarget point_90_contact:=[[190,140,5],[0.707106781,0,0,0.707106781],[0,0,-1,1],[9E+09,9E+09,9E+09,9E+09,9E+09,9E+09]];
    CONST robtarget point_91_contact:=[[194,125,5],[0.707106781,0,0,0.707106781],[0,0,-1,1],[9E+09,9E+09,9E+09,9E+09,9E+09,9E+09]];
    CONST robtarget point_91_clearance:=[[194,125,10],[0.707106781,0,0,0.707106781],[0,0,-1,1],[9E+09,9E+09,9E+09,9E+09,9E+09,9E+09]];
    CONST robtarget point_92_clearance:=[[324,141,10],[0.707106781,0,0,0.707106781],[0,0,-1,1],[9E+09,9E+09,9E+09,9E+09,9E+09,9E+09]];
    CONST robtarget point_92_contact:=[[324,141,5],[0.707106781,0,0,0.707106781],[0,0,-1,1],[9E+09,9E+09,9E+09,9E+09,9E+09,9E+09]];
    CONST robtarget point_93_contact:=[[317,127,5],[0.707106781,0,0,0.707106781],[0,0,-1,1],[9E+09,9E+09,9E+09,9E+09,9E+09,9E+09]];
    CONST robtarget point_93_clearance:=[[317,127,10],[0.707106781,0,0,0.707106781],[0,0,-1,1],[9E+09,9E+09,9E+09,9E+09,9E+09,9E+09]];
    CONST robtarget point_94_clearance:=[[337,127,10],[0.707106781,0,0,0.707106781],[0,0,-1,1],[9E+09,9E+09,9E+09,9E+09,9E+09,9E+09]];
    CONST robtarget point_94_contact:=[[337,127,5],[0.707106781,0,0,0.707106781],[0,0,-1,1],[9E+09,9E+09,9E+09,9E+09,9E+09,9E+09]];
    CONST robtarget point_95_contact:=[[347,133,5],[0.707106781,0,0,0.707106781],[0,0,-1,1],[9E+09,9E+09,9E+09,9E+09,9E+09,9E+09]];
    CONST robtarget point_95_clearance:=[[347,133,10],[0.707106781,0,0,0.707106781],[0,0,-1,1],[9E+09,9E+09,9E+09,9E+09,9E+09,9E+09]];
    CONST robtarget point_96_clearance:=[[184,129,10],[0.707106781,0,0,0.707106781],[0,0,-1,1],[9E+09,9E+09,9E+09,9E+09,9E+09,9E+09]];
    CONST robtarget point_96_contact:=[[184,129,5],[0.707106781,0,0,0.707106781],[0,0,-1,1],[9E+09,9E+09,9E+09,9E+09,9E+09,9E+09]];
    CONST robtarget point_97_contact:=[[174,151,5],[0.707106781,0,0,0.707106781],[0,0,-1,1],[9E+09,9E+09,9E+09,9E+09,9E+09,9E+09]];
    CONST robtarget point_97_clearance:=[[174,151,10],[0.707106781,0,0,0.707106781],[0,0,-1,1],[9E+09,9E+09,9E+09,9E+09,9E+09,9E+09]];
    CONST robtarget point_98_clearance:=[[391,127,10],[0.707106781,0,0,0.707106781],[-1,-1,0,1],[9E+09,9E+09,9E+09,9E+09,9E+09,9E+09]];
    CONST robtarget point_98_contact:=[[391,127,5],[0.707106781,0,0,0.707106781],[-1,-1,0,1],[9E+09,9E+09,9E+09,9E+09,9E+09,9E+09]];
    CONST robtarget point_99_contact:=[[380,144,5],[0.707106781,0,0,0.707106781],[-1,-1,0,1],[9E+09,9E+09,9E+09,9E+09,9E+09,9E+09]];
    CONST robtarget point_99_clearance:=[[380,144,10],[0.707106781,0,0,0.707106781],[-1,-1,0,1],[9E+09,9E+09,9E+09,9E+09,9E+09,9E+09]];
    CONST robtarget point_100_clearance:=[[347,132,10],[0.707106781,0,0,0.707106781],[0,0,-1,1],[9E+09,9E+09,9E+09,9E+09,9E+09,9E+09]];
    CONST robtarget point_100_contact:=[[347,132,5],[0.707106781,0,0,0.707106781],[0,0,-1,1],[9E+09,9E+09,9E+09,9E+09,9E+09,9E+09]];
    CONST robtarget point_101_contact:=[[357,131,5],[0.707106781,0,0,0.707106781],[-1,-1,0,1],[9E+09,9E+09,9E+09,9E+09,9E+09,9E+09]];
    CONST robtarget point_101_clearance:=[[357,131,10],[0.707106781,0,0,0.707106781],[-1,-1,0,1],[9E+09,9E+09,9E+09,9E+09,9E+09,9E+09]];
    CONST robtarget point_102_clearance:=[[150,146,10],[0.707106781,0,0,0.707106781],[0,0,-1,1],[9E+09,9E+09,9E+09,9E+09,9E+09,9E+09]];
    CONST robtarget point_102_contact:=[[150,146,5],[0.707106781,0,0,0.707106781],[0,0,-1,1],[9E+09,9E+09,9E+09,9E+09,9E+09,9E+09]];
    CONST robtarget point_103_contact:=[[160,130,5],[0.707106781,0,0,0.707106781],[0,0,-1,1],[9E+09,9E+09,9E+09,9E+09,9E+09,9E+09]];
    CONST robtarget point_103_clearance:=[[160,130,10],[0.707106781,0,0,0.707106781],[0,0,-1,1],[9E+09,9E+09,9E+09,9E+09,9E+09,9E+09]];
    CONST robtarget point_104_clearance:=[[373,140,10],[0.707106781,0,0,0.707106781],[-1,-1,0,1],[9E+09,9E+09,9E+09,9E+09,9E+09,9E+09]];
    CONST robtarget point_104_contact:=[[373,140,5],[0.707106781,0,0,0.707106781],[-1,-1,0,1],[9E+09,9E+09,9E+09,9E+09,9E+09,9E+09]];
    CONST robtarget point_105_contact:=[[377,146,5],[0.707106781,0,0,0.707106781],[-1,-1,0,1],[9E+09,9E+09,9E+09,9E+09,9E+09,9E+09]];
    CONST robtarget point_105_clearance:=[[377,146,10],[0.707106781,0,0,0.707106781],[-1,-1,0,1],[9E+09,9E+09,9E+09,9E+09,9E+09,9E+09]];
    CONST robtarget point_106_clearance:=[[346,159,10],[0.707106781,0,0,0.707106781],[0,0,-1,1],[9E+09,9E+09,9E+09,9E+09,9E+09,9E+09]];
    CONST robtarget point_106_contact:=[[346,159,5],[0.707106781,0,0,0.707106781],[0,0,-1,1],[9E+09,9E+09,9E+09,9E+09,9E+09,9E+09]];
    CONST robtarget point_107_contact:=[[324,145,5],[0.707106781,0,0,0.707106781],[0,0,-1,1],[9E+09,9E+09,9E+09,9E+09,9E+09,9E+09]];
    CONST robtarget point_107_clearance:=[[324,145,10],[0.707106781,0,0,0.707106781],[0,0,-1,1],[9E+09,9E+09,9E+09,9E+09,9E+09,9E+09]];
    CONST robtarget point_108_clearance:=[[379,148,10],[0.707106781,0,0,0.707106781],[-1,-1,0,1],[9E+09,9E+09,9E+09,9E+09,9E+09,9E+09]];
    CONST robtarget point_108_contact:=[[379,148,5],[0.707106781,0,0,0.707106781],[-1,-1,0,1],[9E+09,9E+09,9E+09,9E+09,9E+09,9E+09]];
    CONST robtarget point_109_contact:=[[353,159,5],[0.707106781,0,0,0.707106781],[0,0,-1,1],[9E+09,9E+09,9E+09,9E+09,9E+09,9E+09]];
    CONST robtarget point_109_clearance:=[[353,159,10],[0.707106781,0,0,0.707106781],[0,0,-1,1],[9E+09,9E+09,9E+09,9E+09,9E+09,9E+09]];
    CONST robtarget point_110_clearance:=[[146,159,10],[0.707106781,0,0,0.707106781],[0,0,-1,1],[9E+09,9E+09,9E+09,9E+09,9E+09,9E+09]];
    CONST robtarget point_110_contact:=[[146,159,5],[0.707106781,0,0,0.707106781],[0,0,-1,1],[9E+09,9E+09,9E+09,9E+09,9E+09,9E+09]];
    CONST robtarget point_111_contact:=[[149,147,5],[0.707106781,0,0,0.707106781],[0,0,-1,1],[9E+09,9E+09,9E+09,9E+09,9E+09,9E+09]];
    CONST robtarget point_111_clearance:=[[149,147,10],[0.707106781,0,0,0.707106781],[0,0,-1,1],[9E+09,9E+09,9E+09,9E+09,9E+09,9E+09]];
    CONST robtarget point_112_clearance:=[[190,160,10],[0.707106781,0,0,0.707106781],[0,0,-1,1],[9E+09,9E+09,9E+09,9E+09,9E+09,9E+09]];
    CONST robtarget point_112_contact:=[[190,160,5],[0.707106781,0,0,0.707106781],[0,0,-1,1],[9E+09,9E+09,9E+09,9E+09,9E+09,9E+09]];
    CONST robtarget point_113_contact:=[[190,148,5],[0.707106781,0,0,0.707106781],[0,0,-1,1],[9E+09,9E+09,9E+09,9E+09,9E+09,9E+09]];
    CONST robtarget point_113_clearance:=[[190,148,10],[0.707106781,0,0,0.707106781],[0,0,-1,1],[9E+09,9E+09,9E+09,9E+09,9E+09,9E+09]];
    CONST robtarget point_114_clearance:=[[174,152,10],[0.707106781,0,0,0.707106781],[0,0,-1,1],[9E+09,9E+09,9E+09,9E+09,9E+09,9E+09]];
    CONST robtarget point_114_contact:=[[174,152,5],[0.707106781,0,0,0.707106781],[0,0,-1,1],[9E+09,9E+09,9E+09,9E+09,9E+09,9E+09]];
    CONST robtarget point_115_contact:=[[179,175,5],[0.707106781,0,0,0.707106781],[0,0,-1,1],[9E+09,9E+09,9E+09,9E+09,9E+09,9E+09]];
    CONST robtarget point_115_clearance:=[[179,175,10],[0.707106781,0,0,0.707106781],[0,0,-1,1],[9E+09,9E+09,9E+09,9E+09,9E+09,9E+09]];
    CONST robtarget point_116_clearance:=[[249,159,10],[0.707106781,0,0,0.707106781],[0,0,-1,1],[9E+09,9E+09,9E+09,9E+09,9E+09,9E+09]];
    CONST robtarget point_116_contact:=[[249,159,5],[0.707106781,0,0,0.707106781],[0,0,-1,1],[9E+09,9E+09,9E+09,9E+09,9E+09,9E+09]];
    CONST robtarget point_117_contact:=[[247,153,5],[0.707106781,0,0,0.707106781],[0,0,-1,1],[9E+09,9E+09,9E+09,9E+09,9E+09,9E+09]];
    CONST robtarget point_117_clearance:=[[247,153,10],[0.707106781,0,0,0.707106781],[0,0,-1,1],[9E+09,9E+09,9E+09,9E+09,9E+09,9E+09]];
    CONST robtarget point_118_clearance:=[[243,167,10],[0.707106781,0,0,0.707106781],[0,0,-1,1],[9E+09,9E+09,9E+09,9E+09,9E+09,9E+09]];
    CONST robtarget point_118_contact:=[[243,167,5],[0.707106781,0,0,0.707106781],[0,0,-1,1],[9E+09,9E+09,9E+09,9E+09,9E+09,9E+09]];
    CONST robtarget point_119_contact:=[[248,159,5],[0.707106781,0,0,0.707106781],[0,0,-1,1],[9E+09,9E+09,9E+09,9E+09,9E+09,9E+09]];
    CONST robtarget point_119_clearance:=[[248,159,10],[0.707106781,0,0,0.707106781],[0,0,-1,1],[9E+09,9E+09,9E+09,9E+09,9E+09,9E+09]];
    CONST robtarget point_120_clearance:=[[201,161,10],[0.707106781,0,0,0.707106781],[0,0,-1,1],[9E+09,9E+09,9E+09,9E+09,9E+09,9E+09]];
    CONST robtarget point_120_contact:=[[201,161,5],[0.707106781,0,0,0.707106781],[0,0,-1,1],[9E+09,9E+09,9E+09,9E+09,9E+09,9E+09]];
    CONST robtarget point_121_contact:=[[193,162,5],[0.707106781,0,0,0.707106781],[0,0,-1,1],[9E+09,9E+09,9E+09,9E+09,9E+09,9E+09]];
    CONST robtarget point_121_clearance:=[[193,162,10],[0.707106781,0,0,0.707106781],[0,0,-1,1],[9E+09,9E+09,9E+09,9E+09,9E+09,9E+09]];
    CONST robtarget point_122_clearance:=[[155,163,10],[0.707106781,0,0,0.707106781],[0,0,-1,1],[9E+09,9E+09,9E+09,9E+09,9E+09,9E+09]];
    CONST robtarget point_122_contact:=[[155,163,5],[0.707106781,0,0,0.707106781],[0,0,-1,1],[9E+09,9E+09,9E+09,9E+09,9E+09,9E+09]];
    CONST robtarget point_123_contact:=[[147,162,5],[0.707106781,0,0,0.707106781],[0,0,-1,1],[9E+09,9E+09,9E+09,9E+09,9E+09,9E+09]];
    CONST robtarget point_123_clearance:=[[147,162,10],[0.707106781,0,0,0.707106781],[0,0,-1,1],[9E+09,9E+09,9E+09,9E+09,9E+09,9E+09]];
    CONST robtarget point_124_clearance:=[[281,162,10],[0.707106781,0,0,0.707106781],[0,0,-1,1],[9E+09,9E+09,9E+09,9E+09,9E+09,9E+09]];
    CONST robtarget point_124_contact:=[[281,162,5],[0.707106781,0,0,0.707106781],[0,0,-1,1],[9E+09,9E+09,9E+09,9E+09,9E+09,9E+09]];
    CONST robtarget point_125_contact:=[[261,182,5],[0.707106781,0,0,0.707106781],[0,0,-1,1],[9E+09,9E+09,9E+09,9E+09,9E+09,9E+09]];
    CONST robtarget point_125_clearance:=[[261,182,10],[0.707106781,0,0,0.707106781],[0,0,-1,1],[9E+09,9E+09,9E+09,9E+09,9E+09,9E+09]];
    CONST robtarget point_126_clearance:=[[189,181,10],[0.707106781,0,0,0.707106781],[0,0,-1,1],[9E+09,9E+09,9E+09,9E+09,9E+09,9E+09]];
    CONST robtarget point_126_contact:=[[189,181,5],[0.707106781,0,0,0.707106781],[0,0,-1,1],[9E+09,9E+09,9E+09,9E+09,9E+09,9E+09]];
    CONST robtarget point_127_contact:=[[190,162,5],[0.707106781,0,0,0.707106781],[0,0,-1,1],[9E+09,9E+09,9E+09,9E+09,9E+09,9E+09]];
    CONST robtarget point_127_clearance:=[[190,162,10],[0.707106781,0,0,0.707106781],[0,0,-1,1],[9E+09,9E+09,9E+09,9E+09,9E+09,9E+09]];
    CONST robtarget point_128_clearance:=[[191,164,10],[0.707106781,0,0,0.707106781],[0,0,-1,1],[9E+09,9E+09,9E+09,9E+09,9E+09,9E+09]];
    CONST robtarget point_128_contact:=[[191,164,5],[0.707106781,0,0,0.707106781],[0,0,-1,1],[9E+09,9E+09,9E+09,9E+09,9E+09,9E+09]];
    CONST robtarget point_129_contact:=[[201,164,5],[0.707106781,0,0,0.707106781],[0,0,-1,1],[9E+09,9E+09,9E+09,9E+09,9E+09,9E+09]];
    CONST robtarget point_129_clearance:=[[201,164,10],[0.707106781,0,0,0.707106781],[0,0,-1,1],[9E+09,9E+09,9E+09,9E+09,9E+09,9E+09]];
    CONST robtarget point_130_clearance:=[[274,181,10],[0.707106781,0,0,0.707106781],[0,0,-1,1],[9E+09,9E+09,9E+09,9E+09,9E+09,9E+09]];
    CONST robtarget point_130_contact:=[[274,181,5],[0.707106781,0,0,0.707106781],[0,0,-1,1],[9E+09,9E+09,9E+09,9E+09,9E+09,9E+09]];
    CONST robtarget point_131_contact:=[[286,167,5],[0.707106781,0,0,0.707106781],[0,0,-1,1],[9E+09,9E+09,9E+09,9E+09,9E+09,9E+09]];
    CONST robtarget point_131_clearance:=[[286,167,10],[0.707106781,0,0,0.707106781],[0,0,-1,1],[9E+09,9E+09,9E+09,9E+09,9E+09,9E+09]];
    CONST robtarget point_132_clearance:=[[286,167,10],[0.707106781,0,0,0.707106781],[0,0,-1,1],[9E+09,9E+09,9E+09,9E+09,9E+09,9E+09]];
    CONST robtarget point_132_contact:=[[286,167,5],[0.707106781,0,0,0.707106781],[0,0,-1,1],[9E+09,9E+09,9E+09,9E+09,9E+09,9E+09]];
    CONST robtarget point_133_contact:=[[320,171,5],[0.707106781,0,0,0.707106781],[0,0,-1,1],[9E+09,9E+09,9E+09,9E+09,9E+09,9E+09]];
    CONST robtarget point_133_clearance:=[[320,171,10],[0.707106781,0,0,0.707106781],[0,0,-1,1],[9E+09,9E+09,9E+09,9E+09,9E+09,9E+09]];
    CONST robtarget point_134_clearance:=[[147,178,10],[0.707106781,0,0,0.707106781],[0,0,-1,1],[9E+09,9E+09,9E+09,9E+09,9E+09,9E+09]];
    CONST robtarget point_134_contact:=[[147,178,5],[0.707106781,0,0,0.707106781],[0,0,-1,1],[9E+09,9E+09,9E+09,9E+09,9E+09,9E+09]];
    CONST robtarget point_135_contact:=[[145,167,5],[0.707106781,0,0,0.707106781],[0,0,-1,1],[9E+09,9E+09,9E+09,9E+09,9E+09,9E+09]];
    CONST robtarget point_135_clearance:=[[145,167,10],[0.707106781,0,0,0.707106781],[0,0,-1,1],[9E+09,9E+09,9E+09,9E+09,9E+09,9E+09]];
    CONST robtarget point_136_clearance:=[[314,169,10],[0.707106781,0,0,0.707106781],[0,0,-1,1],[9E+09,9E+09,9E+09,9E+09,9E+09,9E+09]];
    CONST robtarget point_136_contact:=[[314,169,5],[0.707106781,0,0,0.707106781],[0,0,-1,1],[9E+09,9E+09,9E+09,9E+09,9E+09,9E+09]];
    CONST robtarget point_137_contact:=[[347,179,5],[0.707106781,0,0,0.707106781],[0,0,-1,1],[9E+09,9E+09,9E+09,9E+09,9E+09,9E+09]];
    CONST robtarget point_137_clearance:=[[347,179,10],[0.707106781,0,0,0.707106781],[0,0,-1,1],[9E+09,9E+09,9E+09,9E+09,9E+09,9E+09]];
    CONST robtarget point_138_clearance:=[[178,173,10],[0.707106781,0,0,0.707106781],[0,0,-1,1],[9E+09,9E+09,9E+09,9E+09,9E+09,9E+09]];
    CONST robtarget point_138_contact:=[[178,173,5],[0.707106781,0,0,0.707106781],[0,0,-1,1],[9E+09,9E+09,9E+09,9E+09,9E+09,9E+09]];
    CONST robtarget point_139_contact:=[[188,183,5],[0.707106781,0,0,0.707106781],[0,0,-1,1],[9E+09,9E+09,9E+09,9E+09,9E+09,9E+09]];
    CONST robtarget point_139_clearance:=[[188,183,10],[0.707106781,0,0,0.707106781],[0,0,-1,1],[9E+09,9E+09,9E+09,9E+09,9E+09,9E+09]];
    CONST robtarget point_140_clearance:=[[348,178,10],[0.707106781,0,0,0.707106781],[0,0,-1,1],[9E+09,9E+09,9E+09,9E+09,9E+09,9E+09]];
    CONST robtarget point_140_contact:=[[348,178,5],[0.707106781,0,0,0.707106781],[0,0,-1,1],[9E+09,9E+09,9E+09,9E+09,9E+09,9E+09]];
    CONST robtarget point_141_contact:=[[389,207,5],[0.707106781,0,0,0.707106781],[-1,-1,0,1],[9E+09,9E+09,9E+09,9E+09,9E+09,9E+09]];
    CONST robtarget point_141_clearance:=[[389,207,10],[0.707106781,0,0,0.707106781],[-1,-1,0,1],[9E+09,9E+09,9E+09,9E+09,9E+09,9E+09]];
    CONST robtarget point_142_clearance:=[[149,183,10],[0.707106781,0,0,0.707106781],[0,0,-1,1],[9E+09,9E+09,9E+09,9E+09,9E+09,9E+09]];
    CONST robtarget point_142_contact:=[[149,183,5],[0.707106781,0,0,0.707106781],[0,0,-1,1],[9E+09,9E+09,9E+09,9E+09,9E+09,9E+09]];
    CONST robtarget point_143_contact:=[[157,180,5],[0.707106781,0,0,0.707106781],[0,0,-1,1],[9E+09,9E+09,9E+09,9E+09,9E+09,9E+09]];
    CONST robtarget point_143_clearance:=[[157,180,10],[0.707106781,0,0,0.707106781],[0,0,-1,1],[9E+09,9E+09,9E+09,9E+09,9E+09,9E+09]];
    CONST robtarget point_144_clearance:=[[262,184,10],[0.707106781,0,0,0.707106781],[0,0,-1,1],[9E+09,9E+09,9E+09,9E+09,9E+09,9E+09]];
    CONST robtarget point_144_contact:=[[262,184,5],[0.707106781,0,0,0.707106781],[0,0,-1,1],[9E+09,9E+09,9E+09,9E+09,9E+09,9E+09]];
    CONST robtarget point_145_contact:=[[274,181,5],[0.707106781,0,0,0.707106781],[0,0,-1,1],[9E+09,9E+09,9E+09,9E+09,9E+09,9E+09]];
    CONST robtarget point_145_clearance:=[[274,181,10],[0.707106781,0,0,0.707106781],[0,0,-1,1],[9E+09,9E+09,9E+09,9E+09,9E+09,9E+09]];
    CONST robtarget point_146_clearance:=[[156,199,10],[0.707106781,0,0,0.707106781],[0,0,-1,1],[9E+09,9E+09,9E+09,9E+09,9E+09,9E+09]];
    CONST robtarget point_146_contact:=[[156,199,5],[0.707106781,0,0,0.707106781],[0,0,-1,1],[9E+09,9E+09,9E+09,9E+09,9E+09,9E+09]];
    CONST robtarget point_147_contact:=[[148,184,5],[0.707106781,0,0,0.707106781],[0,0,-1,1],[9E+09,9E+09,9E+09,9E+09,9E+09,9E+09]];
    CONST robtarget point_147_clearance:=[[148,184,10],[0.707106781,0,0,0.707106781],[0,0,-1,1],[9E+09,9E+09,9E+09,9E+09,9E+09,9E+09]];
    CONST robtarget point_148_clearance:=[[355,196,10],[0.707106781,0,0,0.707106781],[0,-1,0,1],[9E+09,9E+09,9E+09,9E+09,9E+09,9E+09]];
    CONST robtarget point_148_contact:=[[355,196,5],[0.707106781,0,0,0.707106781],[0,-1,0,1],[9E+09,9E+09,9E+09,9E+09,9E+09,9E+09]];
    CONST robtarget point_149_contact:=[[331,187,5],[0.707106781,0,0,0.707106781],[0,0,-1,1],[9E+09,9E+09,9E+09,9E+09,9E+09,9E+09]];
    CONST robtarget point_149_clearance:=[[331,187,10],[0.707106781,0,0,0.707106781],[0,0,-1,1],[9E+09,9E+09,9E+09,9E+09,9E+09,9E+09]];
    CONST robtarget point_150_clearance:=[[163,192,10],[0.707106781,0,0,0.707106781],[0,0,-1,1],[9E+09,9E+09,9E+09,9E+09,9E+09,9E+09]];
    CONST robtarget point_150_contact:=[[163,192,5],[0.707106781,0,0,0.707106781],[0,0,-1,1],[9E+09,9E+09,9E+09,9E+09,9E+09,9E+09]];
    CONST robtarget point_151_contact:=[[158,198,5],[0.707106781,0,0,0.707106781],[0,0,-1,1],[9E+09,9E+09,9E+09,9E+09,9E+09,9E+09]];
    CONST robtarget point_151_clearance:=[[158,198,10],[0.707106781,0,0,0.707106781],[0,0,-1,1],[9E+09,9E+09,9E+09,9E+09,9E+09,9E+09]];
    CONST robtarget point_152_clearance:=[[331,190,10],[0.707106781,0,0,0.707106781],[0,0,-1,1],[9E+09,9E+09,9E+09,9E+09,9E+09,9E+09]];
    CONST robtarget point_152_contact:=[[331,190,5],[0.707106781,0,0,0.707106781],[0,0,-1,1],[9E+09,9E+09,9E+09,9E+09,9E+09,9E+09]];
    CONST robtarget point_153_contact:=[[358,201,5],[0.707106781,0,0,0.707106781],[-1,-1,0,1],[9E+09,9E+09,9E+09,9E+09,9E+09,9E+09]];
    CONST robtarget point_153_clearance:=[[358,201,10],[0.707106781,0,0,0.707106781],[-1,-1,0,1],[9E+09,9E+09,9E+09,9E+09,9E+09,9E+09]];
    CONST robtarget point_154_clearance:=[[368,206,10],[0.707106781,0,0,0.707106781],[-1,-1,0,1],[9E+09,9E+09,9E+09,9E+09,9E+09,9E+09]];
    CONST robtarget point_154_contact:=[[368,206,5],[0.707106781,0,0,0.707106781],[-1,-1,0,1],[9E+09,9E+09,9E+09,9E+09,9E+09,9E+09]];
    CONST robtarget point_155_contact:=[[355,197,5],[0.707106781,0,0,0.707106781],[0,-1,0,1],[9E+09,9E+09,9E+09,9E+09,9E+09,9E+09]];
    CONST robtarget point_155_clearance:=[[355,197,10],[0.707106781,0,0,0.707106781],[0,-1,0,1],[9E+09,9E+09,9E+09,9E+09,9E+09,9E+09]];
    CONST robtarget point_156_clearance:=[[160,201,10],[0.707106781,0,0,0.707106781],[0,0,-1,1],[9E+09,9E+09,9E+09,9E+09,9E+09,9E+09]];
    CONST robtarget point_156_contact:=[[160,201,5],[0.707106781,0,0,0.707106781],[0,0,-1,1],[9E+09,9E+09,9E+09,9E+09,9E+09,9E+09]];
    CONST robtarget point_157_contact:=[[166,197,5],[0.707106781,0,0,0.707106781],[0,0,-1,1],[9E+09,9E+09,9E+09,9E+09,9E+09,9E+09]];
    CONST robtarget point_157_clearance:=[[166,197,10],[0.707106781,0,0,0.707106781],[0,0,-1,1],[9E+09,9E+09,9E+09,9E+09,9E+09,9E+09]];
    CONST robtarget point_158_clearance:=[[173,214,10],[0.707106781,0,0,0.707106781],[0,0,-1,1],[9E+09,9E+09,9E+09,9E+09,9E+09,9E+09]];
    CONST robtarget point_158_contact:=[[173,214,5],[0.707106781,0,0,0.707106781],[0,0,-1,1],[9E+09,9E+09,9E+09,9E+09,9E+09,9E+09]];
    CONST robtarget point_159_contact:=[[158,201,5],[0.707106781,0,0,0.707106781],[0,0,-1,1],[9E+09,9E+09,9E+09,9E+09,9E+09,9E+09]];
    CONST robtarget point_159_clearance:=[[158,201,10],[0.707106781,0,0,0.707106781],[0,0,-1,1],[9E+09,9E+09,9E+09,9E+09,9E+09,9E+09]];
    CONST robtarget point_160_clearance:=[[177,202,10],[0.707106781,0,0,0.707106781],[0,0,-1,1],[9E+09,9E+09,9E+09,9E+09,9E+09,9E+09]];
    CONST robtarget point_160_contact:=[[177,202,5],[0.707106781,0,0,0.707106781],[0,0,-1,1],[9E+09,9E+09,9E+09,9E+09,9E+09,9E+09]];
    CONST robtarget point_161_contact:=[[176,212,5],[0.707106781,0,0,0.707106781],[0,0,-1,1],[9E+09,9E+09,9E+09,9E+09,9E+09,9E+09]];
    CONST robtarget point_161_clearance:=[[176,212,10],[0.707106781,0,0,0.707106781],[0,0,-1,1],[9E+09,9E+09,9E+09,9E+09,9E+09,9E+09]];
    CONST robtarget point_162_clearance:=[[358,202,10],[0.707106781,0,0,0.707106781],[-1,-1,0,1],[9E+09,9E+09,9E+09,9E+09,9E+09,9E+09]];
    CONST robtarget point_162_contact:=[[358,202,5],[0.707106781,0,0,0.707106781],[-1,-1,0,1],[9E+09,9E+09,9E+09,9E+09,9E+09,9E+09]];
    CONST robtarget point_163_contact:=[[366,208,5],[0.707106781,0,0,0.707106781],[-1,-1,0,1],[9E+09,9E+09,9E+09,9E+09,9E+09,9E+09]];
    CONST robtarget point_163_clearance:=[[366,208,10],[0.707106781,0,0,0.707106781],[-1,-1,0,1],[9E+09,9E+09,9E+09,9E+09,9E+09,9E+09]];
    CONST robtarget point_164_clearance:=[[173,204,10],[0.707106781,0,0,0.707106781],[0,0,-1,1],[9E+09,9E+09,9E+09,9E+09,9E+09,9E+09]];
    CONST robtarget point_164_contact:=[[173,204,5],[0.707106781,0,0,0.707106781],[0,0,-1,1],[9E+09,9E+09,9E+09,9E+09,9E+09,9E+09]];
    CONST robtarget point_165_contact:=[[174,211,5],[0.707106781,0,0,0.707106781],[0,0,-1,1],[9E+09,9E+09,9E+09,9E+09,9E+09,9E+09]];
    CONST robtarget point_165_clearance:=[[174,211,10],[0.707106781,0,0,0.707106781],[0,0,-1,1],[9E+09,9E+09,9E+09,9E+09,9E+09,9E+09]];
    CONST robtarget point_166_clearance:=[[177,215,10],[0.707106781,0,0,0.707106781],[0,0,-1,1],[9E+09,9E+09,9E+09,9E+09,9E+09,9E+09]];
    CONST robtarget point_166_contact:=[[177,215,5],[0.707106781,0,0,0.707106781],[0,0,-1,1],[9E+09,9E+09,9E+09,9E+09,9E+09,9E+09]];
    CONST robtarget point_167_contact:=[[178,208,5],[0.707106781,0,0,0.707106781],[0,0,-1,1],[9E+09,9E+09,9E+09,9E+09,9E+09,9E+09]];
    CONST robtarget point_167_clearance:=[[178,208,10],[0.707106781,0,0,0.707106781],[0,0,-1,1],[9E+09,9E+09,9E+09,9E+09,9E+09,9E+09]];
    CONST robtarget point_168_clearance:=[[388,208,10],[0.707106781,0,0,0.707106781],[-1,-1,0,1],[9E+09,9E+09,9E+09,9E+09,9E+09,9E+09]];
    CONST robtarget point_168_contact:=[[388,208,5],[0.707106781,0,0,0.707106781],[-1,-1,0,1],[9E+09,9E+09,9E+09,9E+09,9E+09,9E+09]];
    CONST robtarget point_169_contact:=[[389,242,5],[0.707106781,0,0,0.707106781],[-1,-1,0,1],[9E+09,9E+09,9E+09,9E+09,9E+09,9E+09]];
    CONST robtarget point_169_clearance:=[[389,242,10],[0.707106781,0,0,0.707106781],[-1,-1,0,1],[9E+09,9E+09,9E+09,9E+09,9E+09,9E+09]];
    CONST robtarget point_170_clearance:=[[197,223,10],[0.707106781,0,0,0.707106781],[0,0,-1,1],[9E+09,9E+09,9E+09,9E+09,9E+09,9E+09]];
    CONST robtarget point_170_contact:=[[197,223,5],[0.707106781,0,0,0.707106781],[0,0,-1,1],[9E+09,9E+09,9E+09,9E+09,9E+09,9E+09]];
    CONST robtarget point_171_contact:=[[194,209,5],[0.707106781,0,0,0.707106781],[0,0,-1,1],[9E+09,9E+09,9E+09,9E+09,9E+09,9E+09]];
    CONST robtarget point_171_clearance:=[[194,209,10],[0.707106781,0,0,0.707106781],[0,0,-1,1],[9E+09,9E+09,9E+09,9E+09,9E+09,9E+09]];
    CONST robtarget point_172_clearance:=[[252,213,10],[0.707106781,0,0,0.707106781],[0,0,-1,1],[9E+09,9E+09,9E+09,9E+09,9E+09,9E+09]];
    CONST robtarget point_172_contact:=[[252,213,5],[0.707106781,0,0,0.707106781],[0,0,-1,1],[9E+09,9E+09,9E+09,9E+09,9E+09,9E+09]];
    CONST robtarget point_173_contact:=[[238,233,5],[0.707106781,0,0,0.707106781],[0,0,-1,1],[9E+09,9E+09,9E+09,9E+09,9E+09,9E+09]];
    CONST robtarget point_173_clearance:=[[238,233,10],[0.707106781,0,0,0.707106781],[0,0,-1,1],[9E+09,9E+09,9E+09,9E+09,9E+09,9E+09]];
    CONST robtarget point_174_clearance:=[[191,212,10],[0.707106781,0,0,0.707106781],[0,0,-1,1],[9E+09,9E+09,9E+09,9E+09,9E+09,9E+09]];
    CONST robtarget point_174_contact:=[[191,212,5],[0.707106781,0,0,0.707106781],[0,0,-1,1],[9E+09,9E+09,9E+09,9E+09,9E+09,9E+09]];
    CONST robtarget point_175_contact:=[[193,220,5],[0.707106781,0,0,0.707106781],[0,0,-1,1],[9E+09,9E+09,9E+09,9E+09,9E+09,9E+09]];
    CONST robtarget point_175_clearance:=[[193,220,10],[0.707106781,0,0,0.707106781],[0,0,-1,1],[9E+09,9E+09,9E+09,9E+09,9E+09,9E+09]];
    CONST robtarget point_176_clearance:=[[249,232,10],[0.707106781,0,0,0.707106781],[0,0,-1,1],[9E+09,9E+09,9E+09,9E+09,9E+09,9E+09]];
    CONST robtarget point_176_contact:=[[249,232,5],[0.707106781,0,0,0.707106781],[0,0,-1,1],[9E+09,9E+09,9E+09,9E+09,9E+09,9E+09]];
    CONST robtarget point_177_contact:=[[254,212,5],[0.707106781,0,0,0.707106781],[0,0,-1,1],[9E+09,9E+09,9E+09,9E+09,9E+09,9E+09]];
    CONST robtarget point_177_clearance:=[[254,212,10],[0.707106781,0,0,0.707106781],[0,0,-1,1],[9E+09,9E+09,9E+09,9E+09,9E+09,9E+09]];
    CONST robtarget point_178_clearance:=[[394,214,10],[0.707106781,0,0,0.707106781],[-1,-1,0,1],[9E+09,9E+09,9E+09,9E+09,9E+09,9E+09]];
    CONST robtarget point_178_contact:=[[394,214,5],[0.707106781,0,0,0.707106781],[-1,-1,0,1],[9E+09,9E+09,9E+09,9E+09,9E+09,9E+09]];
    CONST robtarget point_179_contact:=[[412,238,5],[0.707106781,0,0,0.707106781],[-1,-1,0,1],[9E+09,9E+09,9E+09,9E+09,9E+09,9E+09]];
    CONST robtarget point_179_clearance:=[[412,238,10],[0.707106781,0,0,0.707106781],[-1,-1,0,1],[9E+09,9E+09,9E+09,9E+09,9E+09,9E+09]];
    CONST robtarget point_180_clearance:=[[192,222,10],[0.707106781,0,0,0.707106781],[0,0,-1,1],[9E+09,9E+09,9E+09,9E+09,9E+09,9E+09]];
    CONST robtarget point_180_contact:=[[192,222,5],[0.707106781,0,0,0.707106781],[0,0,-1,1],[9E+09,9E+09,9E+09,9E+09,9E+09,9E+09]];
    CONST robtarget point_181_contact:=[[177,215,5],[0.707106781,0,0,0.707106781],[0,0,-1,1],[9E+09,9E+09,9E+09,9E+09,9E+09,9E+09]];
    CONST robtarget point_181_clearance:=[[177,215,10],[0.707106781,0,0,0.707106781],[0,0,-1,1],[9E+09,9E+09,9E+09,9E+09,9E+09,9E+09]];
    CONST robtarget point_182_clearance:=[[391,242,10],[0.707106781,0,0,0.707106781],[-1,-1,0,1],[9E+09,9E+09,9E+09,9E+09,9E+09,9E+09]];
    CONST robtarget point_182_contact:=[[391,242,5],[0.707106781,0,0,0.707106781],[-1,-1,0,1],[9E+09,9E+09,9E+09,9E+09,9E+09,9E+09]];
    CONST robtarget point_183_contact:=[[394,216,5],[0.707106781,0,0,0.707106781],[-1,-1,0,1],[9E+09,9E+09,9E+09,9E+09,9E+09,9E+09]];
    CONST robtarget point_183_clearance:=[[394,216,10],[0.707106781,0,0,0.707106781],[-1,-1,0,1],[9E+09,9E+09,9E+09,9E+09,9E+09,9E+09]];
    CONST robtarget point_184_clearance:=[[206,225,10],[0.707106781,0,0,0.707106781],[0,0,-1,1],[9E+09,9E+09,9E+09,9E+09,9E+09,9E+09]];
    CONST robtarget point_184_contact:=[[206,225,5],[0.707106781,0,0,0.707106781],[0,0,-1,1],[9E+09,9E+09,9E+09,9E+09,9E+09,9E+09]];
    CONST robtarget point_185_contact:=[[196,223,5],[0.707106781,0,0,0.707106781],[0,0,-1,1],[9E+09,9E+09,9E+09,9E+09,9E+09,9E+09]];
    CONST robtarget point_185_clearance:=[[196,223,10],[0.707106781,0,0,0.707106781],[0,0,-1,1],[9E+09,9E+09,9E+09,9E+09,9E+09,9E+09]];
    CONST robtarget point_186_clearance:=[[224,248,10],[0.707106781,0,0,0.707106781],[0,0,-1,1],[9E+09,9E+09,9E+09,9E+09,9E+09,9E+09]];
    CONST robtarget point_186_contact:=[[224,248,5],[0.707106781,0,0,0.707106781],[0,0,-1,1],[9E+09,9E+09,9E+09,9E+09,9E+09,9E+09]];
    CONST robtarget point_187_contact:=[[206,226,5],[0.707106781,0,0,0.707106781],[0,0,-1,1],[9E+09,9E+09,9E+09,9E+09,9E+09,9E+09]];
    CONST robtarget point_187_clearance:=[[206,226,10],[0.707106781,0,0,0.707106781],[0,0,-1,1],[9E+09,9E+09,9E+09,9E+09,9E+09,9E+09]];
    CONST robtarget point_188_clearance:=[[242,238,10],[0.707106781,0,0,0.707106781],[0,0,-1,1],[9E+09,9E+09,9E+09,9E+09,9E+09,9E+09]];
    CONST robtarget point_188_contact:=[[242,238,5],[0.707106781,0,0,0.707106781],[0,0,-1,1],[9E+09,9E+09,9E+09,9E+09,9E+09,9E+09]];
    CONST robtarget point_189_contact:=[[248,232,5],[0.707106781,0,0,0.707106781],[0,0,-1,1],[9E+09,9E+09,9E+09,9E+09,9E+09,9E+09]];
    CONST robtarget point_189_clearance:=[[248,232,10],[0.707106781,0,0,0.707106781],[0,0,-1,1],[9E+09,9E+09,9E+09,9E+09,9E+09,9E+09]];
    CONST robtarget point_190_clearance:=[[411,237,10],[0.707106781,0,0,0.707106781],[-1,-1,0,1],[9E+09,9E+09,9E+09,9E+09,9E+09,9E+09]];
    CONST robtarget point_190_contact:=[[411,237,5],[0.707106781,0,0,0.707106781],[-1,-1,0,1],[9E+09,9E+09,9E+09,9E+09,9E+09,9E+09]];
    CONST robtarget point_191_contact:=[[410,287,5],[0.707106781,0,0,0.707106781],[-1,-1,0,1],[9E+09,9E+09,9E+09,9E+09,9E+09,9E+09]];
    CONST robtarget point_191_clearance:=[[410,287,10],[0.707106781,0,0,0.707106781],[-1,-1,0,1],[9E+09,9E+09,9E+09,9E+09,9E+09,9E+09]];
    CONST robtarget point_192_clearance:=[[414,239,10],[0.707106781,0,0,0.707106781],[-1,-1,0,1],[9E+09,9E+09,9E+09,9E+09,9E+09,9E+09]];
    CONST robtarget point_192_contact:=[[414,239,5],[0.707106781,0,0,0.707106781],[-1,-1,0,1],[9E+09,9E+09,9E+09,9E+09,9E+09,9E+09]];
    CONST robtarget point_193_contact:=[[435,285,5],[0.707106781,0,0,0.707106781],[-1,-1,0,1],[9E+09,9E+09,9E+09,9E+09,9E+09,9E+09]];
    CONST robtarget point_193_clearance:=[[435,285,10],[0.707106781,0,0,0.707106781],[-1,-1,0,1],[9E+09,9E+09,9E+09,9E+09,9E+09,9E+09]];
    CONST robtarget point_194_clearance:=[[231,268,10],[0.707106781,0,0,0.707106781],[0,0,-1,1],[9E+09,9E+09,9E+09,9E+09,9E+09,9E+09]];
    CONST robtarget point_194_contact:=[[231,268,5],[0.707106781,0,0,0.707106781],[0,0,-1,1],[9E+09,9E+09,9E+09,9E+09,9E+09,9E+09]];
    CONST robtarget point_195_contact:=[[220,243,5],[0.707106781,0,0,0.707106781],[0,0,-1,1],[9E+09,9E+09,9E+09,9E+09,9E+09,9E+09]];
    CONST robtarget point_195_clearance:=[[220,243,10],[0.707106781,0,0,0.707106781],[0,0,-1,1],[9E+09,9E+09,9E+09,9E+09,9E+09,9E+09]];
    CONST robtarget point_196_clearance:=[[412,286,10],[0.707106781,0,0,0.707106781],[-1,-1,0,1],[9E+09,9E+09,9E+09,9E+09,9E+09,9E+09]];
    CONST robtarget point_196_contact:=[[412,286,5],[0.707106781,0,0,0.707106781],[-1,-1,0,1],[9E+09,9E+09,9E+09,9E+09,9E+09,9E+09]];
    CONST robtarget point_197_contact:=[[415,243,5],[0.707106781,0,0,0.707106781],[-1,-1,0,1],[9E+09,9E+09,9E+09,9E+09,9E+09,9E+09]];
    CONST robtarget point_197_clearance:=[[415,243,10],[0.707106781,0,0,0.707106781],[-1,-1,0,1],[9E+09,9E+09,9E+09,9E+09,9E+09,9E+09]];
    CONST robtarget point_198_clearance:=[[303,259,10],[0.707106781,0,0,0.707106781],[0,0,-1,1],[9E+09,9E+09,9E+09,9E+09,9E+09,9E+09]];
    CONST robtarget point_198_contact:=[[303,259,5],[0.707106781,0,0,0.707106781],[0,0,-1,1],[9E+09,9E+09,9E+09,9E+09,9E+09,9E+09]];
    CONST robtarget point_199_contact:=[[291,259,5],[0.707106781,0,0,0.707106781],[0,0,-1,1],[9E+09,9E+09,9E+09,9E+09,9E+09,9E+09]];
    CONST robtarget point_199_clearance:=[[291,259,10],[0.707106781,0,0,0.707106781],[0,0,-1,1],[9E+09,9E+09,9E+09,9E+09,9E+09,9E+09]];
    CONST robtarget point_200_clearance:=[[291,259,10],[0.707106781,0,0,0.707106781],[0,0,-1,1],[9E+09,9E+09,9E+09,9E+09,9E+09,9E+09]];
    CONST robtarget point_200_contact:=[[291,259,5],[0.707106781,0,0,0.707106781],[0,0,-1,1],[9E+09,9E+09,9E+09,9E+09,9E+09,9E+09]];
    CONST robtarget point_201_contact:=[[278,291,5],[0.707106781,0,0,0.707106781],[0,0,-1,1],[9E+09,9E+09,9E+09,9E+09,9E+09,9E+09]];
    CONST robtarget point_201_clearance:=[[278,291,10],[0.707106781,0,0,0.707106781],[0,0,-1,1],[9E+09,9E+09,9E+09,9E+09,9E+09,9E+09]];
    CONST robtarget point_202_clearance:=[[323,273,10],[0.707106781,0,0,0.707106781],[0,0,-1,1],[9E+09,9E+09,9E+09,9E+09,9E+09,9E+09]];
    CONST robtarget point_202_contact:=[[323,273,5],[0.707106781,0,0,0.707106781],[0,0,-1,1],[9E+09,9E+09,9E+09,9E+09,9E+09,9E+09]];
    CONST robtarget point_203_contact:=[[304,259,5],[0.707106781,0,0,0.707106781],[0,0,-1,1],[9E+09,9E+09,9E+09,9E+09,9E+09,9E+09]];
    CONST robtarget point_203_clearance:=[[304,259,10],[0.707106781,0,0,0.707106781],[0,0,-1,1],[9E+09,9E+09,9E+09,9E+09,9E+09,9E+09]];
    CONST robtarget point_204_clearance:=[[243,322,10],[0.707106781,0,0,0.707106781],[0,0,-1,1],[9E+09,9E+09,9E+09,9E+09,9E+09,9E+09]];
    CONST robtarget point_204_contact:=[[243,322,5],[0.707106781,0,0,0.707106781],[0,0,-1,1],[9E+09,9E+09,9E+09,9E+09,9E+09,9E+09]];
    CONST robtarget point_205_contact:=[[232,266,5],[0.707106781,0,0,0.707106781],[0,0,-1,1],[9E+09,9E+09,9E+09,9E+09,9E+09,9E+09]];
    CONST robtarget point_205_clearance:=[[232,266,10],[0.707106781,0,0,0.707106781],[0,0,-1,1],[9E+09,9E+09,9E+09,9E+09,9E+09,9E+09]];
    CONST robtarget point_206_clearance:=[[328,279,10],[0.707106781,0,0,0.707106781],[0,0,-1,1],[9E+09,9E+09,9E+09,9E+09,9E+09,9E+09]];
    CONST robtarget point_206_contact:=[[328,279,5],[0.707106781,0,0,0.707106781],[0,0,-1,1],[9E+09,9E+09,9E+09,9E+09,9E+09,9E+09]];
    CONST robtarget point_207_contact:=[[323,274,5],[0.707106781,0,0,0.707106781],[0,0,-1,1],[9E+09,9E+09,9E+09,9E+09,9E+09,9E+09]];
    CONST robtarget point_207_clearance:=[[323,274,10],[0.707106781,0,0,0.707106781],[0,0,-1,1],[9E+09,9E+09,9E+09,9E+09,9E+09,9E+09]];
    CONST robtarget point_208_clearance:=[[336,300,10],[0.707106781,0,0,0.707106781],[0,0,-1,1],[9E+09,9E+09,9E+09,9E+09,9E+09,9E+09]];
    CONST robtarget point_208_contact:=[[336,300,5],[0.707106781,0,0,0.707106781],[0,0,-1,1],[9E+09,9E+09,9E+09,9E+09,9E+09,9E+09]];
    CONST robtarget point_209_contact:=[[328,278,5],[0.707106781,0,0,0.707106781],[0,0,-1,1],[9E+09,9E+09,9E+09,9E+09,9E+09,9E+09]];
    CONST robtarget point_209_clearance:=[[328,278,10],[0.707106781,0,0,0.707106781],[0,0,-1,1],[9E+09,9E+09,9E+09,9E+09,9E+09,9E+09]];
    CONST robtarget point_210_clearance:=[[435,285,10],[0.707106781,0,0,0.707106781],[-1,-1,0,1],[9E+09,9E+09,9E+09,9E+09,9E+09,9E+09]];
    CONST robtarget point_210_contact:=[[435,285,5],[0.707106781,0,0,0.707106781],[-1,-1,0,1],[9E+09,9E+09,9E+09,9E+09,9E+09,9E+09]];
    CONST robtarget point_211_contact:=[[432,318,5],[0.707106781,0,0,0.707106781],[-1,-1,0,1],[9E+09,9E+09,9E+09,9E+09,9E+09,9E+09]];
    CONST robtarget point_211_clearance:=[[432,318,10],[0.707106781,0,0,0.707106781],[-1,-1,0,1],[9E+09,9E+09,9E+09,9E+09,9E+09,9E+09]];
    CONST robtarget point_212_clearance:=[[438,289,10],[0.707106781,0,0,0.707106781],[-1,-1,0,1],[9E+09,9E+09,9E+09,9E+09,9E+09,9E+09]];
    CONST robtarget point_212_contact:=[[438,289,5],[0.707106781,0,0,0.707106781],[-1,-1,0,1],[9E+09,9E+09,9E+09,9E+09,9E+09,9E+09]];
    CONST robtarget point_213_contact:=[[444,307,5],[0.707106781,0,0,0.707106781],[-1,-1,0,1],[9E+09,9E+09,9E+09,9E+09,9E+09,9E+09]];
    CONST robtarget point_213_clearance:=[[444,307,10],[0.707106781,0,0,0.707106781],[-1,-1,0,1],[9E+09,9E+09,9E+09,9E+09,9E+09,9E+09]];
    CONST robtarget point_214_clearance:=[[278,291,10],[0.707106781,0,0,0.707106781],[0,0,-1,1],[9E+09,9E+09,9E+09,9E+09,9E+09,9E+09]];
    CONST robtarget point_214_contact:=[[278,291,5],[0.707106781,0,0,0.707106781],[0,0,-1,1],[9E+09,9E+09,9E+09,9E+09,9E+09,9E+09]];
    CONST robtarget point_215_contact:=[[286,313,5],[0.707106781,0,0,0.707106781],[0,0,-1,1],[9E+09,9E+09,9E+09,9E+09,9E+09,9E+09]];
    CONST robtarget point_215_clearance:=[[286,313,10],[0.707106781,0,0,0.707106781],[0,0,-1,1],[9E+09,9E+09,9E+09,9E+09,9E+09,9E+09]];
    CONST robtarget point_216_clearance:=[[435,313,10],[0.707106781,0,0,0.707106781],[-1,-1,0,1],[9E+09,9E+09,9E+09,9E+09,9E+09,9E+09]];
    CONST robtarget point_216_contact:=[[435,313,5],[0.707106781,0,0,0.707106781],[-1,-1,0,1],[9E+09,9E+09,9E+09,9E+09,9E+09,9E+09]];
    CONST robtarget point_217_contact:=[[437,292,5],[0.707106781,0,0,0.707106781],[-1,-1,0,1],[9E+09,9E+09,9E+09,9E+09,9E+09,9E+09]];
    CONST robtarget point_217_clearance:=[[437,292,10],[0.707106781,0,0,0.707106781],[-1,-1,0,1],[9E+09,9E+09,9E+09,9E+09,9E+09,9E+09]];
    CONST robtarget point_218_clearance:=[[333,333,10],[0.707106781,0,0,0.707106781],[0,0,-1,1],[9E+09,9E+09,9E+09,9E+09,9E+09,9E+09]];
    CONST robtarget point_218_contact:=[[333,333,5],[0.707106781,0,0,0.707106781],[0,0,-1,1],[9E+09,9E+09,9E+09,9E+09,9E+09,9E+09]];
    CONST robtarget point_219_contact:=[[334,301,5],[0.707106781,0,0,0.707106781],[0,0,-1,1],[9E+09,9E+09,9E+09,9E+09,9E+09,9E+09]];
    CONST robtarget point_219_clearance:=[[334,301,10],[0.707106781,0,0,0.707106781],[0,0,-1,1],[9E+09,9E+09,9E+09,9E+09,9E+09,9E+09]];
    CONST robtarget point_220_clearance:=[[444,307,10],[0.707106781,0,0,0.707106781],[-1,-1,0,1],[9E+09,9E+09,9E+09,9E+09,9E+09,9E+09]];
    CONST robtarget point_220_contact:=[[444,307,5],[0.707106781,0,0,0.707106781],[-1,-1,0,1],[9E+09,9E+09,9E+09,9E+09,9E+09,9E+09]];
    CONST robtarget point_221_contact:=[[435,316,5],[0.707106781,0,0,0.707106781],[-1,-1,0,1],[9E+09,9E+09,9E+09,9E+09,9E+09,9E+09]];
    CONST robtarget point_221_clearance:=[[435,316,10],[0.707106781,0,0,0.707106781],[-1,-1,0,1],[9E+09,9E+09,9E+09,9E+09,9E+09,9E+09]];
    CONST robtarget point_222_clearance:=[[287,312,10],[0.707106781,0,0,0.707106781],[0,0,-1,1],[9E+09,9E+09,9E+09,9E+09,9E+09,9E+09]];
    CONST robtarget point_222_contact:=[[287,312,5],[0.707106781,0,0,0.707106781],[0,0,-1,1],[9E+09,9E+09,9E+09,9E+09,9E+09,9E+09]];
    CONST robtarget point_223_contact:=[[305,327,5],[0.707106781,0,0,0.707106781],[0,0,-1,1],[9E+09,9E+09,9E+09,9E+09,9E+09,9E+09]];
    CONST robtarget point_223_clearance:=[[305,327,10],[0.707106781,0,0,0.707106781],[0,0,-1,1],[9E+09,9E+09,9E+09,9E+09,9E+09,9E+09]];
    CONST robtarget point_224_clearance:=[[434,317,10],[0.707106781,0,0,0.707106781],[-1,-1,0,1],[9E+09,9E+09,9E+09,9E+09,9E+09,9E+09]];
    CONST robtarget point_224_contact:=[[434,317,5],[0.707106781,0,0,0.707106781],[-1,-1,0,1],[9E+09,9E+09,9E+09,9E+09,9E+09,9E+09]];
    CONST robtarget point_225_contact:=[[352,388,5],[0.707106781,0,0,0.707106781],[0,0,-1,1],[9E+09,9E+09,9E+09,9E+09,9E+09,9E+09]];
    CONST robtarget point_225_clearance:=[[352,388,10],[0.707106781,0,0,0.707106781],[0,0,-1,1],[9E+09,9E+09,9E+09,9E+09,9E+09,9E+09]];
    CONST robtarget point_226_clearance:=[[255,329,10],[0.707106781,0,0,0.707106781],[0,0,-1,1],[9E+09,9E+09,9E+09,9E+09,9E+09,9E+09]];
    CONST robtarget point_226_contact:=[[255,329,5],[0.707106781,0,0,0.707106781],[0,0,-1,1],[9E+09,9E+09,9E+09,9E+09,9E+09,9E+09]];
    CONST robtarget point_227_contact:=[[240,322,5],[0.707106781,0,0,0.707106781],[0,0,-1,1],[9E+09,9E+09,9E+09,9E+09,9E+09,9E+09]];
    CONST robtarget point_227_clearance:=[[240,322,10],[0.707106781,0,0,0.707106781],[0,0,-1,1],[9E+09,9E+09,9E+09,9E+09,9E+09,9E+09]];
    CONST robtarget point_228_clearance:=[[263,326,10],[0.707106781,0,0,0.707106781],[0,0,-1,1],[9E+09,9E+09,9E+09,9E+09,9E+09,9E+09]];
    CONST robtarget point_228_contact:=[[263,326,5],[0.707106781,0,0,0.707106781],[0,0,-1,1],[9E+09,9E+09,9E+09,9E+09,9E+09,9E+09]];
    CONST robtarget point_229_contact:=[[255,329,5],[0.707106781,0,0,0.707106781],[0,0,-1,1],[9E+09,9E+09,9E+09,9E+09,9E+09,9E+09]];
    CONST robtarget point_229_clearance:=[[255,329,10],[0.707106781,0,0,0.707106781],[0,0,-1,1],[9E+09,9E+09,9E+09,9E+09,9E+09,9E+09]];
    CONST robtarget point_230_clearance:=[[283,346,10],[0.707106781,0,0,0.707106781],[0,0,-1,1],[9E+09,9E+09,9E+09,9E+09,9E+09,9E+09]];
    CONST robtarget point_230_contact:=[[283,346,5],[0.707106781,0,0,0.707106781],[0,0,-1,1],[9E+09,9E+09,9E+09,9E+09,9E+09,9E+09]];
    CONST robtarget point_231_contact:=[[262,327,5],[0.707106781,0,0,0.707106781],[0,0,-1,1],[9E+09,9E+09,9E+09,9E+09,9E+09,9E+09]];
    CONST robtarget point_231_clearance:=[[262,327,10],[0.707106781,0,0,0.707106781],[0,0,-1,1],[9E+09,9E+09,9E+09,9E+09,9E+09,9E+09]];
    CONST robtarget point_232_clearance:=[[302,326,10],[0.707106781,0,0,0.707106781],[0,0,-1,1],[9E+09,9E+09,9E+09,9E+09,9E+09,9E+09]];
    CONST robtarget point_232_contact:=[[302,326,5],[0.707106781,0,0,0.707106781],[0,0,-1,1],[9E+09,9E+09,9E+09,9E+09,9E+09,9E+09]];
    CONST robtarget point_233_contact:=[[306,344,5],[0.707106781,0,0,0.707106781],[0,0,-1,1],[9E+09,9E+09,9E+09,9E+09,9E+09,9E+09]];
    CONST robtarget point_233_clearance:=[[306,344,10],[0.707106781,0,0,0.707106781],[0,0,-1,1],[9E+09,9E+09,9E+09,9E+09,9E+09,9E+09]];
    CONST robtarget point_234_clearance:=[[341,379,10],[0.707106781,0,0,0.707106781],[0,0,-1,1],[9E+09,9E+09,9E+09,9E+09,9E+09,9E+09]];
    CONST robtarget point_234_contact:=[[341,379,5],[0.707106781,0,0,0.707106781],[0,0,-1,1],[9E+09,9E+09,9E+09,9E+09,9E+09,9E+09]];
    CONST robtarget point_235_contact:=[[332,335,5],[0.707106781,0,0,0.707106781],[0,0,-1,1],[9E+09,9E+09,9E+09,9E+09,9E+09,9E+09]];
    CONST robtarget point_235_clearance:=[[332,335,10],[0.707106781,0,0,0.707106781],[0,0,-1,1],[9E+09,9E+09,9E+09,9E+09,9E+09,9E+09]];
    CONST robtarget point_236_clearance:=[[293,353,10],[0.707106781,0,0,0.707106781],[0,0,-1,1],[9E+09,9E+09,9E+09,9E+09,9E+09,9E+09]];
    CONST robtarget point_236_contact:=[[293,353,5],[0.707106781,0,0,0.707106781],[0,0,-1,1],[9E+09,9E+09,9E+09,9E+09,9E+09,9E+09]];
    CONST robtarget point_237_contact:=[[285,345,5],[0.707106781,0,0,0.707106781],[0,0,-1,1],[9E+09,9E+09,9E+09,9E+09,9E+09,9E+09]];
    CONST robtarget point_237_clearance:=[[285,345,10],[0.707106781,0,0,0.707106781],[0,0,-1,1],[9E+09,9E+09,9E+09,9E+09,9E+09,9E+09]];
    CONST robtarget point_238_clearance:=[[307,344,10],[0.707106781,0,0,0.707106781],[0,0,-1,1],[9E+09,9E+09,9E+09,9E+09,9E+09,9E+09]];
    CONST robtarget point_238_contact:=[[307,344,5],[0.707106781,0,0,0.707106781],[0,0,-1,1],[9E+09,9E+09,9E+09,9E+09,9E+09,9E+09]];
    CONST robtarget point_239_contact:=[[297,357,5],[0.707106781,0,0,0.707106781],[0,0,-1,1],[9E+09,9E+09,9E+09,9E+09,9E+09,9E+09]];
    CONST robtarget point_239_clearance:=[[297,357,10],[0.707106781,0,0,0.707106781],[0,0,-1,1],[9E+09,9E+09,9E+09,9E+09,9E+09,9E+09]];
    CONST robtarget point_240_clearance:=[[285,360,10],[0.707106781,0,0,0.707106781],[0,0,-1,1],[9E+09,9E+09,9E+09,9E+09,9E+09,9E+09]];
    CONST robtarget point_240_contact:=[[285,360,5],[0.707106781,0,0,0.707106781],[0,0,-1,1],[9E+09,9E+09,9E+09,9E+09,9E+09,9E+09]];
    CONST robtarget point_241_contact:=[[292,353,5],[0.707106781,0,0,0.707106781],[0,0,-1,1],[9E+09,9E+09,9E+09,9E+09,9E+09,9E+09]];
    CONST robtarget point_241_clearance:=[[292,353,10],[0.707106781,0,0,0.707106781],[0,0,-1,1],[9E+09,9E+09,9E+09,9E+09,9E+09,9E+09]];
    CONST robtarget point_242_clearance:=[[297,357,10],[0.707106781,0,0,0.707106781],[0,0,-1,1],[9E+09,9E+09,9E+09,9E+09,9E+09,9E+09]];
    CONST robtarget point_242_contact:=[[297,357,5],[0.707106781,0,0,0.707106781],[0,0,-1,1],[9E+09,9E+09,9E+09,9E+09,9E+09,9E+09]];
    CONST robtarget point_243_contact:=[[298,362,5],[0.707106781,0,0,0.707106781],[0,0,-1,1],[9E+09,9E+09,9E+09,9E+09,9E+09,9E+09]];
    CONST robtarget point_243_clearance:=[[298,362,10],[0.707106781,0,0,0.707106781],[0,0,-1,1],[9E+09,9E+09,9E+09,9E+09,9E+09,9E+09]];
    CONST robtarget point_244_clearance:=[[287,368,10],[0.707106781,0,0,0.707106781],[0,0,-1,1],[9E+09,9E+09,9E+09,9E+09,9E+09,9E+09]];
    CONST robtarget point_244_contact:=[[287,368,5],[0.707106781,0,0,0.707106781],[0,0,-1,1],[9E+09,9E+09,9E+09,9E+09,9E+09,9E+09]];
    CONST robtarget point_245_contact:=[[286,361,5],[0.707106781,0,0,0.707106781],[0,0,-1,1],[9E+09,9E+09,9E+09,9E+09,9E+09,9E+09]];
    CONST robtarget point_245_clearance:=[[286,361,10],[0.707106781,0,0,0.707106781],[0,0,-1,1],[9E+09,9E+09,9E+09,9E+09,9E+09,9E+09]];
    CONST robtarget point_246_clearance:=[[299,362,10],[0.707106781,0,0,0.707106781],[0,0,-1,1],[9E+09,9E+09,9E+09,9E+09,9E+09,9E+09]];
    CONST robtarget point_246_contact:=[[299,362,5],[0.707106781,0,0,0.707106781],[0,0,-1,1],[9E+09,9E+09,9E+09,9E+09,9E+09,9E+09]];
    CONST robtarget point_247_contact:=[[307,373,5],[0.707106781,0,0,0.707106781],[0,0,-1,1],[9E+09,9E+09,9E+09,9E+09,9E+09,9E+09]];
    CONST robtarget point_247_clearance:=[[307,373,10],[0.707106781,0,0,0.707106781],[0,0,-1,1],[9E+09,9E+09,9E+09,9E+09,9E+09,9E+09]];
    CONST robtarget point_248_clearance:=[[297,374,10],[0.707106781,0,0,0.707106781],[0,0,-1,1],[9E+09,9E+09,9E+09,9E+09,9E+09,9E+09]];
    CONST robtarget point_248_contact:=[[297,374,5],[0.707106781,0,0,0.707106781],[0,0,-1,1],[9E+09,9E+09,9E+09,9E+09,9E+09,9E+09]];
    CONST robtarget point_249_contact:=[[286,369,5],[0.707106781,0,0,0.707106781],[0,0,-1,1],[9E+09,9E+09,9E+09,9E+09,9E+09,9E+09]];
    CONST robtarget point_249_clearance:=[[286,369,10],[0.707106781,0,0,0.707106781],[0,0,-1,1],[9E+09,9E+09,9E+09,9E+09,9E+09,9E+09]];
    CONST robtarget point_250_clearance:=[[304,370,10],[0.707106781,0,0,0.707106781],[0,0,-1,1],[9E+09,9E+09,9E+09,9E+09,9E+09,9E+09]];
    CONST robtarget point_250_contact:=[[304,370,5],[0.707106781,0,0,0.707106781],[0,0,-1,1],[9E+09,9E+09,9E+09,9E+09,9E+09,9E+09]];
    CONST robtarget point_251_contact:=[[307,377,5],[0.707106781,0,0,0.707106781],[0,0,-1,1],[9E+09,9E+09,9E+09,9E+09,9E+09,9E+09]];
    CONST robtarget point_251_clearance:=[[307,377,10],[0.707106781,0,0,0.707106781],[0,0,-1,1],[9E+09,9E+09,9E+09,9E+09,9E+09,9E+09]];
    CONST robtarget point_252_clearance:=[[303,383,10],[0.707106781,0,0,0.707106781],[0,0,-1,1],[9E+09,9E+09,9E+09,9E+09,9E+09,9E+09]];
    CONST robtarget point_252_contact:=[[303,383,5],[0.707106781,0,0,0.707106781],[0,0,-1,1],[9E+09,9E+09,9E+09,9E+09,9E+09,9E+09]];
    CONST robtarget point_253_contact:=[[303,375,5],[0.707106781,0,0,0.707106781],[0,0,-1,1],[9E+09,9E+09,9E+09,9E+09,9E+09,9E+09]];
    CONST robtarget point_253_clearance:=[[303,375,10],[0.707106781,0,0,0.707106781],[0,0,-1,1],[9E+09,9E+09,9E+09,9E+09,9E+09,9E+09]];
    CONST robtarget point_254_clearance:=[[350,387,10],[0.707106781,0,0,0.707106781],[0,0,-1,1],[9E+09,9E+09,9E+09,9E+09,9E+09,9E+09]];
    CONST robtarget point_254_contact:=[[350,387,5],[0.707106781,0,0,0.707106781],[0,0,-1,1],[9E+09,9E+09,9E+09,9E+09,9E+09,9E+09]];
    CONST robtarget point_255_contact:=[[341,377,5],[0.707106781,0,0,0.707106781],[0,0,-1,1],[9E+09,9E+09,9E+09,9E+09,9E+09,9E+09]];
    CONST robtarget point_255_clearance:=[[341,377,10],[0.707106781,0,0,0.707106781],[0,0,-1,1],[9E+09,9E+09,9E+09,9E+09,9E+09,9E+09]];



